LIN {X 177.96, Y 27.59, Z 0.00, A 0, B 0, C 0} C_DIS
LIN {X 177.78, Y 27.40, Z 0.00, A 0, B 0, C 0} C_DIS
LIN {X 177.60, Y 27.22, Z 0.00, A 0, B 0, C 0} C_DIS
LIN {X 177.41, Y 27.05, Z 0.00, A 0, B 0, C 0} C_DIS
LIN {X 177.23, Y 26.88, Z 0.00, A 0, B 0, C 0} C_DIS
LIN {X 177.05, Y 26.69, Z 0.00, A 0, B 0, C 0} C_DIS
LIN {X 176.88, Y 26.50, Z 0.00, A 0, B 0, C 0} C_DIS
LIN {X 176.71, Y 26.29, Z 0.00, A 0, B 0, C 0} C_DIS
LIN {X 176.55, Y 26.07, Z 0.00, A 0, B 0, C 0} C_DIS
LIN {X 176.39, Y 25.84, Z 0.00, A 0, B 0, C 0} C_DIS
LIN {X 176.24, Y 25.61, Z 0.00, A 0, B 0, C 0} C_DIS
LIN {X 176.09, Y 25.38, Z 0.00, A 0, B 0, C 0} C_DIS
LIN {X 175.93, Y 25.14, Z 0.00, A 0, B 0, C 0} C_DIS
LIN {X 175.78, Y 24.91, Z 0.00, A 0, B 0, C 0} C_DIS
LIN {X 175.63, Y 24.68, Z 0.00, A 0, B 0, C 0} C_DIS
LIN {X 175.47, Y 24.45, Z 0.00, A 0, B 0, C 0} C_DIS
LIN {X 175.32, Y 24.21, Z 0.00, A 0, B 0, C 0} C_DIS
LIN {X 175.17, Y 23.98, Z 0.00, A 0, B 0, C 0} C_DIS
LIN {X 175.01, Y 23.75, Z 0.00, A 0, B 0, C 0} C_DIS
LIN {X 174.86, Y 23.52, Z 0.00, A 0, B 0, C 0} C_DIS
LIN {X 174.71, Y 23.29, Z 0.00, A 0, B 0, C 0} C_DIS
LIN {X 174.55, Y 23.05, Z 0.00, A 0, B 0, C 0} C_DIS
LIN {X 174.40, Y 22.82, Z 0.00, A 0, B 0, C 0} C_DIS
LIN {X 174.24, Y 22.59, Z 0.00, A 0, B 0, C 0} C_DIS
LIN {X 174.09, Y 22.36, Z 0.00, A 0, B 0, C 0} C_DIS
LIN {X 173.94, Y 22.13, Z 0.00, A 0, B 0, C 0} C_DIS
LIN {X 173.78, Y 21.90, Z 0.00, A 0, B 0, C 0} C_DIS
LIN {X 173.63, Y 21.66, Z 0.00, A 0, B 0, C 0} C_DIS
LIN {X 173.48, Y 21.43, Z 0.00, A 0, B 0, C 0} C_DIS
LIN {X 173.32, Y 21.20, Z 0.00, A 0, B 0, C 0} C_DIS
LIN {X 173.17, Y 20.97, Z 0.00, A 0, B 0, C 0} C_DIS
LIN {X 173.01, Y 20.74, Z 0.00, A 0, B 0, C 0} C_DIS
LIN {X 172.86, Y 20.51, Z 0.00, A 0, B 0, C 0} C_DIS
LIN {X 172.71, Y 20.28, Z 0.00, A 0, B 0, C 0} C_DIS
LIN {X 172.55, Y 20.04, Z 0.00, A 0, B 0, C 0} C_DIS
LIN {X 172.40, Y 19.81, Z 0.00, A 0, B 0, C 0} C_DIS
LIN {X 172.24, Y 19.58, Z 0.00, A 0, B 0, C 0} C_DIS
LIN {X 172.09, Y 19.35, Z 0.00, A 0, B 0, C 0} C_DIS
LIN {X 171.94, Y 19.12, Z 0.00, A 0, B 0, C 0} C_DIS
LIN {X 171.78, Y 18.89, Z 0.00, A 0, B 0, C 0} C_DIS
LIN {X 171.63, Y 18.65, Z 0.00, A 0, B 0, C 0} C_DIS
LIN {X 171.48, Y 18.42, Z 0.00, A 0, B 0, C 0} C_DIS
LIN {X 171.32, Y 18.19, Z 0.00, A 0, B 0, C 0} C_DIS
LIN {X 171.17, Y 17.96, Z 0.00, A 0, B 0, C 0} C_DIS
LIN {X 171.01, Y 17.73, Z 0.00, A 0, B 0, C 0} C_DIS
LIN {X 170.86, Y 17.49, Z 0.00, A 0, B 0, C 0} C_DIS
LIN {X 170.71, Y 17.26, Z 0.00, A 0, B 0, C 0} C_DIS
LIN {X 170.55, Y 17.03, Z 0.00, A 0, B 0, C 0} C_DIS
LIN {X 170.40, Y 16.80, Z 0.00, A 0, B 0, C 0} C_DIS
LIN {X 170.25, Y 16.57, Z 0.00, A 0, B 0, C 0} C_DIS
LIN {X 170.09, Y 16.33, Z 0.00, A 0, B 0, C 0} C_DIS
LIN {X 169.94, Y 16.10, Z 0.00, A 0, B 0, C 0} C_DIS
LIN {X 169.78, Y 15.87, Z 0.00, A 0, B 0, C 0} C_DIS
LIN {X 169.63, Y 15.64, Z 0.00, A 0, B 0, C 0} C_DIS
LIN {X 169.48, Y 15.41, Z 0.00, A 0, B 0, C 0} C_DIS
LIN {X 169.32, Y 15.18, Z 0.00, A 0, B 0, C 0} C_DIS
LIN {X 169.17, Y 14.94, Z 0.00, A 0, B 0, C 0} C_DIS
LIN {X 169.02, Y 14.71, Z 0.00, A 0, B 0, C 0} C_DIS
LIN {X 168.86, Y 14.48, Z 0.00, A 0, B 0, C 0} C_DIS
LIN {X 168.71, Y 14.25, Z 0.00, A 0, B 0, C 0} C_DIS
LIN {X 168.55, Y 14.02, Z 0.00, A 0, B 0, C 0} C_DIS
LIN {X 168.40, Y 13.79, Z 0.00, A 0, B 0, C 0} C_DIS
LIN {X 168.25, Y 13.55, Z 0.00, A 0, B 0, C 0} C_DIS
LIN {X 168.09, Y 13.32, Z 0.00, A 0, B 0, C 0} C_DIS
LIN {X 167.94, Y 13.09, Z 0.00, A 0, B 0, C 0} C_DIS
LIN {X 167.79, Y 12.86, Z 0.00, A 0, B 0, C 0} C_DIS
LIN {X 167.63, Y 12.63, Z 0.00, A 0, B 0, C 0} C_DIS
LIN {X 167.48, Y 12.40, Z 0.00, A 0, B 0, C 0} C_DIS
LIN {X 167.32, Y 12.17, Z 0.00, A 0, B 0, C 0} C_DIS
LIN {X 167.17, Y 11.93, Z 0.00, A 0, B 0, C 0} C_DIS
LIN {X 167.02, Y 11.70, Z 0.00, A 0, B 0, C 0} C_DIS
LIN {X 166.86, Y 11.47, Z 0.00, A 0, B 0, C 0} C_DIS
LIN {X 166.71, Y 11.24, Z 0.00, A 0, B 0, C 0} C_DIS
LIN {X 166.55, Y 11.01, Z 0.00, A 0, B 0, C 0} C_DIS
LIN {X 166.40, Y 10.78, Z 0.00, A 0, B 0, C 0} C_DIS
LIN {X 166.25, Y 10.54, Z 0.00, A 0, B 0, C 0} C_DIS
LIN {X 166.09, Y 10.31, Z 0.00, A 0, B 0, C 0} C_DIS
LIN {X 165.94, Y 10.08, Z 0.00, A 0, B 0, C 0} C_DIS
LIN {X 165.79, Y 9.85, Z 0.00, A 0, B 0, C 0} C_DIS
LIN {X 165.63, Y 9.62, Z 0.00, A 0, B 0, C 0} C_DIS
LIN {X 165.48, Y 9.38, Z 0.00, A 0, B 0, C 0} C_DIS
LIN {X 165.33, Y 9.15, Z 0.00, A 0, B 0, C 0} C_DIS
LIN {X 165.17, Y 8.92, Z 0.00, A 0, B 0, C 0} C_DIS
LIN {X 165.02, Y 8.68, Z 0.00, A 0, B 0, C 0} C_DIS
LIN {X 164.87, Y 8.45, Z 0.00, A 0, B 0, C 0} C_DIS
LIN {X 164.71, Y 8.22, Z 0.00, A 0, B 0, C 0} C_DIS
LIN {X 164.56, Y 7.99, Z 0.00, A 0, B 0, C 0} C_DIS
LIN {X 164.40, Y 7.76, Z 0.00, A 0, B 0, C 0} C_DIS
LIN {X 164.24, Y 7.54, Z 0.00, A 0, B 0, C 0} C_DIS
LIN {X 164.08, Y 7.33, Z 0.00, A 0, B 0, C 0} C_DIS
LIN {X 163.91, Y 7.13, Z 0.00, A 0, B 0, C 0} C_DIS
LIN {X 163.73, Y 6.94, Z 0.00, A 0, B 0, C 0} C_DIS
LIN {X 163.54, Y 6.77, Z 0.00, A 0, B 0, C 0} C_DIS
LIN {X 163.36, Y 6.60, Z 0.00, A 0, B 0, C 0} C_DIS
LIN {X 163.17, Y 6.42, Z 0.00, A 0, B 0, C 0} C_DIS
LIN {X 163.00, Y 6.23, Z 0.00, A 0, B 0, C 0} C_DIS
LIN {X 162.83, Y 6.02, Z 0.00, A 0, B 0, C 0} C_DIS
LIN {X 162.67, Y 5.80, Z 0.00, A 0, B 0, C 0} C_DIS
LIN {X 162.51, Y 5.58, Z 0.00, A 0, B 0, C 0} C_DIS
LIN {X 162.34, Y 5.37, Z 0.00, A 0, B 0, C 0} C_DIS
LIN {X 162.17, Y 5.17, Z 0.00, A 0, B 0, C 0} C_DIS
LIN {X 162.00, Y 4.98, Z 0.00, A 0, B 0, C 0} C_DIS
LIN {X 161.81, Y 4.80, Z 0.00, A 0, B 0, C 0} C_DIS
LIN {X 161.62, Y 4.64, Z 0.00, A 0, B 0, C 0} C_DIS
LIN {X 161.43, Y 4.51, Z 0.00, A 0, B 0, C 0} C_DIS
LIN {X 161.23, Y 4.38, Z 0.00, A 0, B 0, C 0} C_DIS
LIN {X 161.03, Y 4.23, Z 0.00, A 0, B 0, C 0} C_DIS
LIN {X 160.84, Y 4.07, Z 0.00, A 0, B 0, C 0} C_DIS
LIN {X 160.66, Y 3.89, Z 0.00, A 0, B 0, C 0} C_DIS
LIN {X 160.48, Y 3.70, Z 0.00, A 0, B 0, C 0} C_DIS
LIN {X 160.30, Y 3.52, Z 0.00, A 0, B 0, C 0} C_DIS
LIN {X 160.12, Y 3.33, Z 0.00, A 0, B 0, C 0} C_DIS
LIN {X 159.94, Y 3.15, Z 0.00, A 0, B 0, C 0} C_DIS
LIN {X 159.76, Y 2.97, Z 0.00, A 0, B 0, C 0} C_DIS
LIN {X 159.58, Y 2.79, Z 0.00, A 0, B 0, C 0} C_DIS
LIN {X 159.39, Y 2.63, Z 0.00, A 0, B 0, C 0} C_DIS
LIN {X 159.20, Y 2.49, Z 0.00, A 0, B 0, C 0} C_DIS
LIN {X 158.99, Y 2.39, Z 0.00, A 0, B 0, C 0} C_DIS
LIN {X 158.78, Y 2.31, Z 0.00, A 0, B 0, C 0} C_DIS
LIN {X 158.56, Y 2.25, Z 0.00, A 0, B 0, C 0} C_DIS
LIN {X 158.35, Y 2.17, Z 0.00, A 0, B 0, C 0} C_DIS
LIN {X 158.14, Y 2.09, Z 0.00, A 0, B 0, C 0} C_DIS
LIN {X 157.93, Y 2.00, Z 0.00, A 0, B 0, C 0} C_DIS
LIN {X 157.72, Y 1.92, Z 0.00, A 0, B 0, C 0} C_DIS
LIN {X 157.51, Y 1.85, Z 0.00, A 0, B 0, C 0} C_DIS
LIN {X 157.30, Y 1.78, Z 0.00, A 0, B 0, C 0} C_DIS
LIN {X 157.09, Y 1.69, Z 0.00, A 0, B 0, C 0} C_DIS
LIN {X 156.88, Y 1.57, Z 0.00, A 0, B 0, C 0} C_DIS
LIN {X 156.69, Y 1.44, Z 0.00, A 0, B 0, C 0} C_DIS
LIN {X 156.49, Y 1.31, Z 0.00, A 0, B 0, C 0} C_DIS
LIN {X 156.28, Y 1.21, Z 0.00, A 0, B 0, C 0} C_DIS
LIN {X 156.07, Y 1.14, Z 0.00, A 0, B 0, C 0} C_DIS
LIN {X 155.85, Y 1.06, Z 0.00, A 0, B 0, C 0} C_DIS
LIN {X 155.64, Y 0.98, Z 0.00, A 0, B 0, C 0} C_DIS
LIN {X 155.43, Y 0.89, Z 0.00, A 0, B 0, C 0} C_DIS
LIN {X 155.22, Y 0.84, Z 0.00, A 0, B 0, C 0} C_DIS
LIN {X 155.00, Y 0.82, Z 0.00, A 0, B 0, C 0} C_DIS
LIN {X 154.79, Y 0.81, Z 0.00, A 0, B 0, C 0} C_DIS
LIN {X 154.57, Y 0.81, Z 0.00, A 0, B 0, C 0} C_DIS
LIN {X 154.35, Y 0.81, Z 0.00, A 0, B 0, C 0} C_DIS
LIN {X 154.13, Y 0.81, Z 0.00, A 0, B 0, C 0} C_DIS
LIN {X 153.92, Y 0.81, Z 0.00, A 0, B 0, C 0} C_DIS
LIN {X 153.70, Y 0.82, Z 0.00, A 0, B 0, C 0} C_DIS
LIN {X 153.48, Y 0.82, Z 0.00, A 0, B 0, C 0} C_DIS
LIN {X 153.26, Y 0.82, Z 0.00, A 0, B 0, C 0} C_DIS
LIN {X 153.05, Y 0.81, Z 0.00, A 0, B 0, C 0} C_DIS
LIN {X 152.83, Y 0.81, Z 0.00, A 0, B 0, C 0} C_DIS
LIN {X 152.61, Y 0.81, Z 0.00, A 0, B 0, C 0} C_DIS
LIN {X 152.39, Y 0.81, Z 0.00, A 0, B 0, C 0} C_DIS
LIN {X 152.18, Y 0.81, Z 0.00, A 0, B 0, C 0} C_DIS
LIN {X 151.96, Y 0.81, Z 0.00, A 0, B 0, C 0} C_DIS
LIN {X 151.74, Y 0.81, Z 0.00, A 0, B 0, C 0} C_DIS
LIN {X 151.52, Y 0.81, Z 0.00, A 0, B 0, C 0} C_DIS
LIN {X 151.31, Y 0.81, Z 0.00, A 0, B 0, C 0} C_DIS
LIN {X 151.09, Y 0.81, Z 0.00, A 0, B 0, C 0} C_DIS
LIN {X 150.87, Y 0.81, Z 0.00, A 0, B 0, C 0} C_DIS
LIN {X 150.65, Y 0.81, Z 0.00, A 0, B 0, C 0} C_DIS
LIN {X 150.44, Y 0.81, Z 0.00, A 0, B 0, C 0} C_DIS
LIN {X 150.22, Y 0.81, Z 0.00, A 0, B 0, C 0} C_DIS
LIN {X 150.00, Y 0.81, Z 0.00, A 0, B 0, C 0} C_DIS
LIN {X 149.78, Y 0.81, Z 0.00, A 0, B 0, C 0} C_DIS
LIN {X 149.57, Y 0.81, Z 0.00, A 0, B 0, C 0} C_DIS
LIN {X 149.35, Y 0.81, Z 0.00, A 0, B 0, C 0} C_DIS
LIN {X 149.13, Y 0.81, Z 0.00, A 0, B 0, C 0} C_DIS
LIN {X 148.91, Y 0.81, Z 0.00, A 0, B 0, C 0} C_DIS
LIN {X 148.70, Y 0.81, Z 0.00, A 0, B 0, C 0} C_DIS
LIN {X 148.48, Y 0.81, Z 0.00, A 0, B 0, C 0} C_DIS
LIN {X 148.26, Y 0.81, Z 0.00, A 0, B 0, C 0} C_DIS
LIN {X 148.04, Y 0.81, Z 0.00, A 0, B 0, C 0} C_DIS
LIN {X 147.83, Y 0.81, Z 0.00, A 0, B 0, C 0} C_DIS
LIN {X 147.61, Y 0.81, Z 0.00, A 0, B 0, C 0} C_DIS
LIN {X 147.39, Y 0.81, Z 0.00, A 0, B 0, C 0} C_DIS
LIN {X 147.17, Y 0.81, Z 0.00, A 0, B 0, C 0} C_DIS
LIN {X 146.96, Y 0.81, Z 0.00, A 0, B 0, C 0} C_DIS
LIN {X 146.74, Y 0.81, Z 0.00, A 0, B 0, C 0} C_DIS
LIN {X 146.52, Y 0.81, Z 0.00, A 0, B 0, C 0} C_DIS
LIN {X 146.30, Y 0.81, Z 0.00, A 0, B 0, C 0} C_DIS
LIN {X 146.09, Y 0.81, Z 0.00, A 0, B 0, C 0} C_DIS
LIN {X 145.87, Y 0.81, Z 0.00, A 0, B 0, C 0} C_DIS
LIN {X 145.65, Y 0.81, Z 0.00, A 0, B 0, C 0} C_DIS
LIN {X 145.43, Y 0.81, Z 0.00, A 0, B 0, C 0} C_DIS
LIN {X 145.22, Y 0.81, Z 0.00, A 0, B 0, C 0} C_DIS
LIN {X 145.00, Y 0.81, Z 0.00, A 0, B 0, C 0} C_DIS
LIN {X 144.78, Y 0.81, Z 0.00, A 0, B 0, C 0} C_DIS
LIN {X 144.56, Y 0.81, Z 0.00, A 0, B 0, C 0} C_DIS
LIN {X 144.35, Y 0.81, Z 0.00, A 0, B 0, C 0} C_DIS
LIN {X 144.13, Y 0.81, Z 0.00, A 0, B 0, C 0} C_DIS
LIN {X 143.91, Y 0.81, Z 0.00, A 0, B 0, C 0} C_DIS
LIN {X 143.69, Y 0.81, Z 0.00, A 0, B 0, C 0} C_DIS
LIN {X 143.48, Y 0.81, Z 0.00, A 0, B 0, C 0} C_DIS
LIN {X 143.26, Y 0.81, Z 0.00, A 0, B 0, C 0} C_DIS
LIN {X 143.04, Y 0.81, Z 0.00, A 0, B 0, C 0} C_DIS
LIN {X 142.83, Y 0.81, Z 0.00, A 0, B 0, C 0} C_DIS
LIN {X 142.61, Y 0.81, Z 0.00, A 0, B 0, C 0} C_DIS
LIN {X 142.39, Y 0.81, Z 0.00, A 0, B 0, C 0} C_DIS
LIN {X 142.17, Y 0.81, Z 0.00, A 0, B 0, C 0} C_DIS
LIN {X 141.96, Y 0.81, Z 0.00, A 0, B 0, C 0} C_DIS
LIN {X 141.74, Y 0.81, Z 0.00, A 0, B 0, C 0} C_DIS
LIN {X 141.52, Y 0.81, Z 0.00, A 0, B 0, C 0} C_DIS
LIN {X 141.30, Y 0.81, Z 0.00, A 0, B 0, C 0} C_DIS
LIN {X 141.09, Y 0.81, Z 0.00, A 0, B 0, C 0} C_DIS
LIN {X 140.87, Y 0.81, Z 0.00, A 0, B 0, C 0} C_DIS
LIN {X 140.65, Y 0.81, Z 0.00, A 0, B 0, C 0} C_DIS
LIN {X 140.43, Y 0.81, Z 0.00, A 0, B 0, C 0} C_DIS
LIN {X 140.22, Y 0.81, Z 0.00, A 0, B 0, C 0} C_DIS
LIN {X 140.00, Y 0.81, Z 0.00, A 0, B 0, C 0} C_DIS
LIN {X 139.78, Y 0.81, Z 0.00, A 0, B 0, C 0} C_DIS
LIN {X 139.56, Y 0.81, Z 0.00, A 0, B 0, C 0} C_DIS
LIN {X 139.35, Y 0.81, Z 0.00, A 0, B 0, C 0} C_DIS
LIN {X 139.13, Y 0.81, Z 0.00, A 0, B 0, C 0} C_DIS
LIN {X 138.91, Y 0.81, Z 0.00, A 0, B 0, C 0} C_DIS
LIN {X 138.69, Y 0.81, Z 0.00, A 0, B 0, C 0} C_DIS
LIN {X 138.48, Y 0.81, Z 0.00, A 0, B 0, C 0} C_DIS
LIN {X 138.26, Y 0.81, Z 0.00, A 0, B 0, C 0} C_DIS
LIN {X 138.04, Y 0.81, Z 0.00, A 0, B 0, C 0} C_DIS
LIN {X 137.82, Y 0.81, Z 0.00, A 0, B 0, C 0} C_DIS
LIN {X 137.61, Y 0.81, Z 0.00, A 0, B 0, C 0} C_DIS
LIN {X 137.39, Y 0.81, Z 0.00, A 0, B 0, C 0} C_DIS
LIN {X 137.17, Y 0.81, Z 0.00, A 0, B 0, C 0} C_DIS
LIN {X 136.95, Y 0.81, Z 0.00, A 0, B 0, C 0} C_DIS
LIN {X 136.74, Y 0.81, Z 0.00, A 0, B 0, C 0} C_DIS
LIN {X 136.52, Y 0.81, Z 0.00, A 0, B 0, C 0} C_DIS
LIN {X 136.30, Y 0.81, Z 0.00, A 0, B 0, C 0} C_DIS
LIN {X 136.08, Y 0.81, Z 0.00, A 0, B 0, C 0} C_DIS
LIN {X 135.87, Y 0.81, Z 0.00, A 0, B 0, C 0} C_DIS
LIN {X 135.65, Y 0.81, Z 0.00, A 0, B 0, C 0} C_DIS
LIN {X 135.43, Y 0.82, Z 0.00, A 0, B 0, C 0} C_DIS
LIN {X 135.21, Y 0.82, Z 0.00, A 0, B 0, C 0} C_DIS
LIN {X 135.00, Y 0.81, Z 0.00, A 0, B 0, C 0} C_DIS
LIN {X 134.78, Y 0.81, Z 0.00, A 0, B 0, C 0} C_DIS
LIN {X 134.56, Y 0.81, Z 0.00, A 0, B 0, C 0} C_DIS
LIN {X 134.34, Y 0.81, Z 0.00, A 0, B 0, C 0} C_DIS
LIN {X 134.13, Y 0.80, Z 0.00, A 0, B 0, C 0} C_DIS
LIN {X 133.91, Y 0.81, Z 0.00, A 0, B 0, C 0} C_DIS
LIN {X 133.69, Y 0.82, Z 0.00, A 0, B 0, C 0} C_DIS
LIN {X 133.48, Y 0.85, Z 0.00, A 0, B 0, C 0} C_DIS
LIN {X 133.26, Y 0.90, Z 0.00, A 0, B 0, C 0} C_DIS
LIN {X 133.05, Y 0.98, Z 0.00, A 0, B 0, C 0} C_DIS
LIN {X 132.84, Y 1.06, Z 0.00, A 0, B 0, C 0} C_DIS
LIN {X 132.63, Y 1.14, Z 0.00, A 0, B 0, C 0} C_DIS
LIN {X 132.42, Y 1.26, Z 0.00, A 0, B 0, C 0} C_DIS
LIN {X 132.24, Y 1.42, Z 0.00, A 0, B 0, C 0} C_DIS
LIN {X 132.08, Y 1.65, Z 0.00, A 0, B 0, C 0} C_DIS
LIN {X 131.93, Y 1.89, Z 0.00, A 0, B 0, C 0} C_DIS
LIN {X 131.78, Y 2.13, Z 0.00, A 0, B 0, C 0} C_DIS
LIN {X 131.64, Y 2.37, Z 0.00, A 0, B 0, C 0} C_DIS
LIN {X 131.53, Y 2.64, Z 0.00, A 0, B 0, C 0} C_DIS
LIN {X 131.45, Y 2.95, Z 0.00, A 0, B 0, C 0} C_DIS
LIN {X 131.40, Y 3.28, Z 0.00, A 0, B 0, C 0} C_DIS
LIN {X 131.36, Y 3.60, Z 0.00, A 0, B 0, C 0} C_DIS
LIN {X 131.32, Y 3.93, Z 0.00, A 0, B 0, C 0} C_DIS
LIN {X 131.29, Y 4.25, Z 0.00, A 0, B 0, C 0} C_DIS
LIN {X 131.27, Y 4.57, Z 0.00, A 0, B 0, C 0} C_DIS
LIN {X 131.26, Y 4.89, Z 0.00, A 0, B 0, C 0} C_DIS
LIN {X 131.25, Y 5.22, Z 0.00, A 0, B 0, C 0} C_DIS
LIN {X 131.25, Y 5.55, Z 0.00, A 0, B 0, C 0} C_DIS
LIN {X 131.25, Y 5.88, Z 0.00, A 0, B 0, C 0} C_DIS
LIN {X 131.26, Y 6.21, Z 0.00, A 0, B 0, C 0} C_DIS
LIN {X 131.26, Y 6.53, Z 0.00, A 0, B 0, C 0} C_DIS
LIN {X 131.26, Y 6.86, Z 0.00, A 0, B 0, C 0} C_DIS
LIN {X 131.26, Y 7.19, Z 0.00, A 0, B 0, C 0} C_DIS
LIN {X 131.26, Y 7.52, Z 0.00, A 0, B 0, C 0} C_DIS
LIN {X 131.26, Y 7.85, Z 0.00, A 0, B 0, C 0} C_DIS
LIN {X 131.26, Y 8.17, Z 0.00, A 0, B 0, C 0} C_DIS
LIN {X 131.26, Y 8.50, Z 0.00, A 0, B 0, C 0} C_DIS
LIN {X 131.26, Y 8.83, Z 0.00, A 0, B 0, C 0} C_DIS
LIN {X 131.26, Y 9.16, Z 0.00, A 0, B 0, C 0} C_DIS
LIN {X 131.26, Y 9.49, Z 0.00, A 0, B 0, C 0} C_DIS
LIN {X 131.26, Y 9.81, Z 0.00, A 0, B 0, C 0} C_DIS
LIN {X 131.26, Y 10.14, Z 0.00, A 0, B 0, C 0} C_DIS
LIN {X 131.26, Y 10.47, Z 0.00, A 0, B 0, C 0} C_DIS
LIN {X 131.26, Y 10.80, Z 0.00, A 0, B 0, C 0} C_DIS
LIN {X 131.26, Y 11.12, Z 0.00, A 0, B 0, C 0} C_DIS
LIN {X 131.26, Y 11.45, Z 0.00, A 0, B 0, C 0} C_DIS
LIN {X 131.26, Y 11.78, Z 0.00, A 0, B 0, C 0} C_DIS
LIN {X 131.26, Y 12.11, Z 0.00, A 0, B 0, C 0} C_DIS
LIN {X 131.26, Y 12.43, Z 0.00, A 0, B 0, C 0} C_DIS
LIN {X 131.26, Y 12.76, Z 0.00, A 0, B 0, C 0} C_DIS
LIN {X 131.26, Y 13.09, Z 0.00, A 0, B 0, C 0} C_DIS
LIN {X 131.26, Y 13.42, Z 0.00, A 0, B 0, C 0} C_DIS
LIN {X 131.26, Y 13.75, Z 0.00, A 0, B 0, C 0} C_DIS
LIN {X 131.26, Y 14.07, Z 0.00, A 0, B 0, C 0} C_DIS
LIN {X 131.26, Y 14.40, Z 0.00, A 0, B 0, C 0} C_DIS
LIN {X 131.26, Y 14.73, Z 0.00, A 0, B 0, C 0} C_DIS
LIN {X 131.26, Y 15.06, Z 0.00, A 0, B 0, C 0} C_DIS
LIN {X 131.26, Y 15.38, Z 0.00, A 0, B 0, C 0} C_DIS
LIN {X 131.26, Y 15.71, Z 0.00, A 0, B 0, C 0} C_DIS
LIN {X 131.26, Y 16.04, Z 0.00, A 0, B 0, C 0} C_DIS
LIN {X 131.26, Y 16.37, Z 0.00, A 0, B 0, C 0} C_DIS
LIN {X 131.26, Y 16.69, Z 0.00, A 0, B 0, C 0} C_DIS
LIN {X 131.26, Y 17.02, Z 0.00, A 0, B 0, C 0} C_DIS
LIN {X 131.26, Y 17.35, Z 0.00, A 0, B 0, C 0} C_DIS
LIN {X 131.26, Y 17.68, Z 0.00, A 0, B 0, C 0} C_DIS
LIN {X 131.26, Y 18.01, Z 0.00, A 0, B 0, C 0} C_DIS
LIN {X 131.26, Y 18.33, Z 0.00, A 0, B 0, C 0} C_DIS
LIN {X 131.26, Y 18.66, Z 0.00, A 0, B 0, C 0} C_DIS
LIN {X 131.26, Y 18.99, Z 0.00, A 0, B 0, C 0} C_DIS
LIN {X 131.26, Y 19.32, Z 0.00, A 0, B 0, C 0} C_DIS
LIN {X 131.26, Y 19.64, Z 0.00, A 0, B 0, C 0} C_DIS
LIN {X 131.26, Y 19.97, Z 0.00, A 0, B 0, C 0} C_DIS
LIN {X 131.26, Y 20.30, Z 0.00, A 0, B 0, C 0} C_DIS
LIN {X 131.26, Y 20.63, Z 0.00, A 0, B 0, C 0} C_DIS
LIN {X 131.26, Y 20.95, Z 0.00, A 0, B 0, C 0} C_DIS
LIN {X 131.26, Y 21.28, Z 0.00, A 0, B 0, C 0} C_DIS
LIN {X 131.26, Y 21.61, Z 0.00, A 0, B 0, C 0} C_DIS
LIN {X 131.26, Y 21.94, Z 0.00, A 0, B 0, C 0} C_DIS
LIN {X 131.26, Y 22.27, Z 0.00, A 0, B 0, C 0} C_DIS
LIN {X 131.26, Y 22.59, Z 0.00, A 0, B 0, C 0} C_DIS
LIN {X 131.26, Y 22.92, Z 0.00, A 0, B 0, C 0} C_DIS
LIN {X 131.26, Y 23.25, Z 0.00, A 0, B 0, C 0} C_DIS
LIN {X 131.26, Y 23.58, Z 0.00, A 0, B 0, C 0} C_DIS
LIN {X 131.26, Y 23.90, Z 0.00, A 0, B 0, C 0} C_DIS
LIN {X 131.26, Y 24.23, Z 0.00, A 0, B 0, C 0} C_DIS
LIN {X 131.26, Y 24.56, Z 0.00, A 0, B 0, C 0} C_DIS
LIN {X 131.26, Y 24.89, Z 0.00, A 0, B 0, C 0} C_DIS
LIN {X 131.26, Y 25.21, Z 0.00, A 0, B 0, C 0} C_DIS
LIN {X 131.26, Y 25.54, Z 0.00, A 0, B 0, C 0} C_DIS
LIN {X 131.26, Y 25.87, Z 0.00, A 0, B 0, C 0} C_DIS
LIN {X 131.26, Y 26.20, Z 0.00, A 0, B 0, C 0} C_DIS
LIN {X 131.26, Y 26.53, Z 0.00, A 0, B 0, C 0} C_DIS
LIN {X 131.26, Y 26.85, Z 0.00, A 0, B 0, C 0} C_DIS
LIN {X 131.26, Y 27.18, Z 0.00, A 0, B 0, C 0} C_DIS
LIN {X 131.26, Y 27.51, Z 0.00, A 0, B 0, C 0} C_DIS
LIN {X 131.26, Y 27.84, Z 0.00, A 0, B 0, C 0} C_DIS
LIN {X 131.26, Y 28.16, Z 0.00, A 0, B 0, C 0} C_DIS
LIN {X 131.26, Y 28.49, Z 0.00, A 0, B 0, C 0} C_DIS
LIN {X 131.26, Y 28.82, Z 0.00, A 0, B 0, C 0} C_DIS
LIN {X 131.26, Y 29.15, Z 0.00, A 0, B 0, C 0} C_DIS
LIN {X 131.26, Y 29.48, Z 0.00, A 0, B 0, C 0} C_DIS
LIN {X 131.26, Y 29.80, Z 0.00, A 0, B 0, C 0} C_DIS
LIN {X 131.26, Y 30.13, Z 0.00, A 0, B 0, C 0} C_DIS
LIN {X 131.26, Y 30.46, Z 0.00, A 0, B 0, C 0} C_DIS
LIN {X 131.26, Y 30.79, Z 0.00, A 0, B 0, C 0} C_DIS
LIN {X 131.26, Y 31.11, Z 0.00, A 0, B 0, C 0} C_DIS
LIN {X 131.26, Y 31.44, Z 0.00, A 0, B 0, C 0} C_DIS
LIN {X 131.26, Y 31.77, Z 0.00, A 0, B 0, C 0} C_DIS
LIN {X 131.26, Y 32.10, Z 0.00, A 0, B 0, C 0} C_DIS
LIN {X 131.26, Y 32.42, Z 0.00, A 0, B 0, C 0} C_DIS
LIN {X 131.26, Y 32.75, Z 0.00, A 0, B 0, C 0} C_DIS
LIN {X 131.26, Y 33.08, Z 0.00, A 0, B 0, C 0} C_DIS
LIN {X 131.26, Y 33.41, Z 0.00, A 0, B 0, C 0} C_DIS
LIN {X 131.26, Y 33.74, Z 0.00, A 0, B 0, C 0} C_DIS
LIN {X 131.26, Y 34.06, Z 0.00, A 0, B 0, C 0} C_DIS
LIN {X 131.26, Y 34.39, Z 0.00, A 0, B 0, C 0} C_DIS
LIN {X 131.26, Y 34.72, Z 0.00, A 0, B 0, C 0} C_DIS
LIN {X 131.26, Y 35.05, Z 0.00, A 0, B 0, C 0} C_DIS
LIN {X 131.26, Y 35.37, Z 0.00, A 0, B 0, C 0} C_DIS
LIN {X 131.26, Y 35.70, Z 0.00, A 0, B 0, C 0} C_DIS
LIN {X 131.26, Y 36.03, Z 0.00, A 0, B 0, C 0} C_DIS
LIN {X 131.26, Y 36.36, Z 0.00, A 0, B 0, C 0} C_DIS
LIN {X 131.26, Y 36.69, Z 0.00, A 0, B 0, C 0} C_DIS
LIN {X 131.26, Y 37.01, Z 0.00, A 0, B 0, C 0} C_DIS
LIN {X 131.26, Y 37.34, Z 0.00, A 0, B 0, C 0} C_DIS
LIN {X 131.26, Y 37.67, Z 0.00, A 0, B 0, C 0} C_DIS
LIN {X 131.26, Y 38.00, Z 0.00, A 0, B 0, C 0} C_DIS
LIN {X 131.26, Y 38.32, Z 0.00, A 0, B 0, C 0} C_DIS
LIN {X 131.26, Y 38.65, Z 0.00, A 0, B 0, C 0} C_DIS
LIN {X 131.26, Y 38.98, Z 0.00, A 0, B 0, C 0} C_DIS
LIN {X 131.26, Y 39.31, Z 0.00, A 0, B 0, C 0} C_DIS
LIN {X 131.26, Y 39.63, Z 0.00, A 0, B 0, C 0} C_DIS
LIN {X 131.26, Y 39.96, Z 0.00, A 0, B 0, C 0} C_DIS
LIN {X 131.26, Y 40.29, Z 0.00, A 0, B 0, C 0} C_DIS
LIN {X 131.26, Y 40.62, Z 0.00, A 0, B 0, C 0} C_DIS
LIN {X 131.26, Y 40.95, Z 0.00, A 0, B 0, C 0} C_DIS
LIN {X 131.26, Y 41.27, Z 0.00, A 0, B 0, C 0} C_DIS
LIN {X 131.26, Y 41.60, Z 0.00, A 0, B 0, C 0} C_DIS
LIN {X 131.26, Y 41.93, Z 0.00, A 0, B 0, C 0} C_DIS
LIN {X 131.26, Y 42.26, Z 0.00, A 0, B 0, C 0} C_DIS
LIN {X 131.26, Y 42.58, Z 0.00, A 0, B 0, C 0} C_DIS
LIN {X 131.26, Y 42.91, Z 0.00, A 0, B 0, C 0} C_DIS
LIN {X 131.26, Y 43.24, Z 0.00, A 0, B 0, C 0} C_DIS
LIN {X 131.26, Y 43.57, Z 0.00, A 0, B 0, C 0} C_DIS
LIN {X 131.26, Y 43.89, Z 0.00, A 0, B 0, C 0} C_DIS
LIN {X 131.26, Y 44.22, Z 0.00, A 0, B 0, C 0} C_DIS
LIN {X 131.26, Y 44.55, Z 0.00, A 0, B 0, C 0} C_DIS
LIN {X 131.26, Y 44.88, Z 0.00, A 0, B 0, C 0} C_DIS
LIN {X 131.26, Y 45.21, Z 0.00, A 0, B 0, C 0} C_DIS
LIN {X 131.26, Y 45.53, Z 0.00, A 0, B 0, C 0} C_DIS
LIN {X 131.26, Y 45.86, Z 0.00, A 0, B 0, C 0} C_DIS
LIN {X 131.26, Y 46.19, Z 0.00, A 0, B 0, C 0} C_DIS
LIN {X 131.26, Y 46.52, Z 0.00, A 0, B 0, C 0} C_DIS
LIN {X 131.26, Y 46.84, Z 0.00, A 0, B 0, C 0} C_DIS
LIN {X 131.26, Y 47.17, Z 0.00, A 0, B 0, C 0} C_DIS
LIN {X 131.26, Y 47.50, Z 0.00, A 0, B 0, C 0} C_DIS
LIN {X 131.26, Y 47.83, Z 0.00, A 0, B 0, C 0} C_DIS
LIN {X 131.26, Y 48.16, Z 0.00, A 0, B 0, C 0} C_DIS
LIN {X 131.26, Y 48.48, Z 0.00, A 0, B 0, C 0} C_DIS
LIN {X 131.26, Y 48.81, Z 0.00, A 0, B 0, C 0} C_DIS
LIN {X 131.26, Y 49.14, Z 0.00, A 0, B 0, C 0} C_DIS
LIN {X 131.26, Y 49.47, Z 0.00, A 0, B 0, C 0} C_DIS
LIN {X 131.26, Y 49.79, Z 0.00, A 0, B 0, C 0} C_DIS
LIN {X 131.26, Y 50.12, Z 0.00, A 0, B 0, C 0} C_DIS
LIN {X 131.26, Y 50.45, Z 0.00, A 0, B 0, C 0} C_DIS
LIN {X 131.26, Y 50.78, Z 0.00, A 0, B 0, C 0} C_DIS
LIN {X 131.26, Y 51.10, Z 0.00, A 0, B 0, C 0} C_DIS
LIN {X 131.26, Y 51.43, Z 0.00, A 0, B 0, C 0} C_DIS
LIN {X 131.26, Y 51.76, Z 0.00, A 0, B 0, C 0} C_DIS
LIN {X 131.26, Y 52.09, Z 0.00, A 0, B 0, C 0} C_DIS
LIN {X 131.26, Y 52.42, Z 0.00, A 0, B 0, C 0} C_DIS
LIN {X 131.26, Y 52.74, Z 0.00, A 0, B 0, C 0} C_DIS
LIN {X 131.26, Y 53.07, Z 0.00, A 0, B 0, C 0} C_DIS
LIN {X 131.26, Y 53.40, Z 0.00, A 0, B 0, C 0} C_DIS
LIN {X 131.26, Y 53.73, Z 0.00, A 0, B 0, C 0} C_DIS
LIN {X 131.26, Y 54.05, Z 0.00, A 0, B 0, C 0} C_DIS
LIN {X 131.26, Y 54.38, Z 0.00, A 0, B 0, C 0} C_DIS
LIN {X 131.26, Y 54.71, Z 0.00, A 0, B 0, C 0} C_DIS
LIN {X 131.26, Y 55.04, Z 0.00, A 0, B 0, C 0} C_DIS
LIN {X 131.26, Y 55.36, Z 0.00, A 0, B 0, C 0} C_DIS
LIN {X 131.26, Y 55.69, Z 0.00, A 0, B 0, C 0} C_DIS
LIN {X 131.26, Y 56.02, Z 0.00, A 0, B 0, C 0} C_DIS
LIN {X 131.26, Y 56.35, Z 0.00, A 0, B 0, C 0} C_DIS
LIN {X 131.26, Y 56.68, Z 0.00, A 0, B 0, C 0} C_DIS
LIN {X 131.26, Y 57.00, Z 0.00, A 0, B 0, C 0} C_DIS
LIN {X 131.26, Y 57.33, Z 0.00, A 0, B 0, C 0} C_DIS
LIN {X 131.26, Y 57.66, Z 0.00, A 0, B 0, C 0} C_DIS
LIN {X 131.26, Y 57.99, Z 0.00, A 0, B 0, C 0} C_DIS
LIN {X 131.26, Y 58.31, Z 0.00, A 0, B 0, C 0} C_DIS
LIN {X 131.26, Y 58.64, Z 0.00, A 0, B 0, C 0} C_DIS
LIN {X 131.26, Y 58.97, Z 0.00, A 0, B 0, C 0} C_DIS
LIN {X 131.26, Y 59.30, Z 0.00, A 0, B 0, C 0} C_DIS
LIN {X 131.26, Y 59.63, Z 0.00, A 0, B 0, C 0} C_DIS
LIN {X 131.27, Y 59.95, Z 0.00, A 0, B 0, C 0} C_DIS
LIN {X 131.27, Y 60.28, Z 0.00, A 0, B 0, C 0} C_DIS
LIN {X 131.27, Y 60.61, Z 0.00, A 0, B 0, C 0} C_DIS
LIN {X 131.27, Y 60.94, Z 0.00, A 0, B 0, C 0} C_DIS
LIN {X 131.27, Y 61.26, Z 0.00, A 0, B 0, C 0} C_DIS
LIN {X 131.26, Y 61.59, Z 0.00, A 0, B 0, C 0} C_DIS
LIN {X 131.25, Y 61.92, Z 0.00, A 0, B 0, C 0} C_DIS
LIN {X 131.24, Y 62.25, Z 0.00, A 0, B 0, C 0} C_DIS
LIN {X 131.23, Y 62.57, Z 0.00, A 0, B 0, C 0} C_DIS
LIN {X 131.20, Y 62.90, Z 0.00, A 0, B 0, C 0} C_DIS
LIN {X 131.16, Y 63.22, Z 0.00, A 0, B 0, C 0} C_DIS
LIN {X 131.11, Y 63.53, Z 0.00, A 0, B 0, C 0} C_DIS
LIN {X 131.04, Y 63.85, Z 0.00, A 0, B 0, C 0} C_DIS
LIN {X 130.98, Y 64.17, Z 0.00, A 0, B 0, C 0} C_DIS
LIN {X 130.93, Y 64.48, Z 0.00, A 0, B 0, C 0} C_DIS
LIN {X 130.88, Y 64.80, Z 0.00, A 0, B 0, C 0} C_DIS
LIN {X 130.85, Y 65.13, Z 0.00, A 0, B 0, C 0} C_DIS
LIN {X 130.83, Y 65.45, Z 0.00, A 0, B 0, C 0} C_DIS
LIN {X 130.82, Y 65.78, Z 0.00, A 0, B 0, C 0} C_DIS
LIN {X 130.82, Y 66.11, Z 0.00, A 0, B 0, C 0} C_DIS
LIN {X 130.82, Y 66.43, Z 0.00, A 0, B 0, C 0} C_DIS
LIN {X 130.83, Y 66.76, Z 0.00, A 0, B 0, C 0} C_DIS
LIN {X 130.83, Y 67.09, Z 0.00, A 0, B 0, C 0} C_DIS
LIN {X 130.84, Y 67.42, Z 0.00, A 0, B 0, C 0} C_DIS
LIN {X 130.83, Y 67.75, Z 0.00, A 0, B 0, C 0} C_DIS
LIN {X 130.82, Y 68.07, Z 0.00, A 0, B 0, C 0} C_DIS
LIN {X 130.80, Y 68.40, Z 0.00, A 0, B 0, C 0} C_DIS
LIN {X 130.77, Y 68.72, Z 0.00, A 0, B 0, C 0} C_DIS
LIN {X 130.73, Y 69.04, Z 0.00, A 0, B 0, C 0} C_DIS
LIN {X 130.68, Y 69.36, Z 0.00, A 0, B 0, C 0} C_DIS
LIN {X 130.63, Y 69.68, Z 0.00, A 0, B 0, C 0} C_DIS
LIN {X 130.57, Y 70.00, Z 0.00, A 0, B 0, C 0} C_DIS
LIN {X 130.51, Y 70.31, Z 0.00, A 0, B 0, C 0} C_DIS
LIN {X 130.46, Y 70.63, Z 0.00, A 0, B 0, C 0} C_DIS
LIN {X 130.40, Y 70.95, Z 0.00, A 0, B 0, C 0} C_DIS
LIN {X 130.35, Y 71.27, Z 0.00, A 0, B 0, C 0} C_DIS
LIN {X 130.30, Y 71.59, Z 0.00, A 0, B 0, C 0} C_DIS
LIN {X 130.25, Y 71.90, Z 0.00, A 0, B 0, C 0} C_DIS
LIN {X 130.20, Y 72.22, Z 0.00, A 0, B 0, C 0} C_DIS
LIN {X 130.15, Y 72.54, Z 0.00, A 0, B 0, C 0} C_DIS
LIN {X 130.08, Y 72.85, Z 0.00, A 0, B 0, C 0} C_DIS
LIN {X 130.01, Y 73.16, Z 0.00, A 0, B 0, C 0} C_DIS
LIN {X 129.92, Y 73.46, Z 0.00, A 0, B 0, C 0} C_DIS
LIN {X 129.83, Y 73.76, Z 0.00, A 0, B 0, C 0} C_DIS
LIN {X 129.78, Y 74.08, Z 0.00, A 0, B 0, C 0} C_DIS
LIN {X 129.72, Y 74.39, Z 0.00, A 0, B 0, C 0} C_DIS
LIN {X 129.63, Y 74.69, Z 0.00, A 0, B 0, C 0} C_DIS
LIN {X 129.52, Y 74.97, Z 0.00, A 0, B 0, C 0} C_DIS
LIN {X 129.40, Y 75.25, Z 0.00, A 0, B 0, C 0} C_DIS
LIN {X 129.32, Y 75.55, Z 0.00, A 0, B 0, C 0} C_DIS
LIN {X 129.27, Y 75.87, Z 0.00, A 0, B 0, C 0} C_DIS
LIN {X 129.21, Y 76.19, Z 0.00, A 0, B 0, C 0} C_DIS
LIN {X 129.12, Y 76.49, Z 0.00, A 0, B 0, C 0} C_DIS
LIN {X 129.03, Y 76.78, Z 0.00, A 0, B 0, C 0} C_DIS
LIN {X 128.95, Y 77.09, Z 0.00, A 0, B 0, C 0} C_DIS
LIN {X 128.90, Y 77.41, Z 0.00, A 0, B 0, C 0} C_DIS
LIN {X 128.84, Y 77.72, Z 0.00, A 0, B 0, C 0} C_DIS
LIN {X 128.75, Y 78.02, Z 0.00, A 0, B 0, C 0} C_DIS
LIN {X 128.63, Y 78.29, Z 0.00, A 0, B 0, C 0} C_DIS
LIN {X 128.52, Y 78.58, Z 0.00, A 0, B 0, C 0} C_DIS
LIN {X 128.44, Y 78.88, Z 0.00, A 0, B 0, C 0} C_DIS
LIN {X 128.35, Y 79.18, Z 0.00, A 0, B 0, C 0} C_DIS
LIN {X 128.25, Y 79.47, Z 0.00, A 0, B 0, C 0} C_DIS
LIN {X 128.14, Y 79.75, Z 0.00, A 0, B 0, C 0} C_DIS
LIN {X 128.02, Y 80.02, Z 0.00, A 0, B 0, C 0} C_DIS
LIN {X 127.89, Y 80.29, Z 0.00, A 0, B 0, C 0} C_DIS
LIN {X 127.76, Y 80.56, Z 0.00, A 0, B 0, C 0} C_DIS
LIN {X 127.64, Y 80.83, Z 0.00, A 0, B 0, C 0} C_DIS
LIN {X 127.52, Y 81.10, Z 0.00, A 0, B 0, C 0} C_DIS
LIN {X 127.40, Y 81.38, Z 0.00, A 0, B 0, C 0} C_DIS
LIN {X 127.30, Y 81.66, Z 0.00, A 0, B 0, C 0} C_DIS
LIN {X 127.20, Y 81.95, Z 0.00, A 0, B 0, C 0} C_DIS
LIN {X 127.11, Y 82.25, Z 0.00, A 0, B 0, C 0} C_DIS
LIN {X 127.01, Y 82.54, Z 0.00, A 0, B 0, C 0} C_DIS
LIN {X 126.91, Y 82.83, Z 0.00, A 0, B 0, C 0} C_DIS
LIN {X 126.80, Y 83.11, Z 0.00, A 0, B 0, C 0} C_DIS
LIN {X 126.68, Y 83.38, Z 0.00, A 0, B 0, C 0} C_DIS
LIN {X 126.54, Y 83.64, Z 0.00, A 0, B 0, C 0} C_DIS
LIN {X 126.40, Y 83.89, Z 0.00, A 0, B 0, C 0} C_DIS
LIN {X 126.26, Y 84.13, Z 0.00, A 0, B 0, C 0} C_DIS
LIN {X 126.11, Y 84.36, Z 0.00, A 0, B 0, C 0} C_DIS
LIN {X 125.95, Y 84.59, Z 0.00, A 0, B 0, C 0} C_DIS
LIN {X 125.79, Y 84.82, Z 0.00, A 0, B 0, C 0} C_DIS
LIN {X 125.64, Y 85.06, Z 0.00, A 0, B 0, C 0} C_DIS
LIN {X 125.51, Y 85.31, Z 0.00, A 0, B 0, C 0} C_DIS
LIN {X 125.39, Y 85.59, Z 0.00, A 0, B 0, C 0} C_DIS
LIN {X 125.27, Y 85.87, Z 0.00, A 0, B 0, C 0} C_DIS
LIN {X 125.16, Y 86.15, Z 0.00, A 0, B 0, C 0} C_DIS
LIN {X 125.04, Y 86.43, Z 0.00, A 0, B 0, C 0} C_DIS
LIN {X 124.92, Y 86.70, Z 0.00, A 0, B 0, C 0} C_DIS
LIN {X 124.79, Y 86.95, Z 0.00, A 0, B 0, C 0} C_DIS
LIN {X 124.64, Y 87.20, Z 0.00, A 0, B 0, C 0} C_DIS
LIN {X 124.49, Y 87.43, Z 0.00, A 0, B 0, C 0} C_DIS
LIN {X 124.34, Y 87.67, Z 0.00, A 0, B 0, C 0} C_DIS
LIN {X 124.19, Y 87.90, Z 0.00, A 0, B 0, C 0} C_DIS
LIN {X 124.03, Y 88.13, Z 0.00, A 0, B 0, C 0} C_DIS
LIN {X 123.88, Y 88.37, Z 0.00, A 0, B 0, C 0} C_DIS
LIN {X 123.73, Y 88.60, Z 0.00, A 0, B 0, C 0} C_DIS
LIN {X 123.58, Y 88.83, Z 0.00, A 0, B 0, C 0} C_DIS
LIN {X 123.42, Y 89.06, Z 0.00, A 0, B 0, C 0} C_DIS
LIN {X 123.26, Y 89.27, Z 0.00, A 0, B 0, C 0} C_DIS
LIN {X 123.09, Y 89.48, Z 0.00, A 0, B 0, C 0} C_DIS
LIN {X 122.91, Y 89.67, Z 0.00, A 0, B 0, C 0} C_DIS
LIN {X 122.73, Y 89.85, Z 0.00, A 0, B 0, C 0} C_DIS
LIN {X 122.55, Y 90.03, Z 0.00, A 0, B 0, C 0} C_DIS
LIN {X 122.36, Y 90.20, Z 0.00, A 0, B 0, C 0} C_DIS
LIN {X 122.18, Y 90.38, Z 0.00, A 0, B 0, C 0} C_DIS
LIN {X 122.00, Y 90.57, Z 0.00, A 0, B 0, C 0} C_DIS
LIN {X 121.84, Y 90.78, Z 0.00, A 0, B 0, C 0} C_DIS
LIN {X 121.68, Y 91.01, Z 0.00, A 0, B 0, C 0} C_DIS
LIN {X 121.53, Y 91.24, Z 0.00, A 0, B 0, C 0} C_DIS
LIN {X 121.38, Y 91.48, Z 0.00, A 0, B 0, C 0} C_DIS
LIN {X 121.23, Y 91.71, Z 0.00, A 0, B 0, C 0} C_DIS
LIN {X 121.07, Y 91.93, Z 0.00, A 0, B 0, C 0} C_DIS
LIN {X 120.89, Y 92.13, Z 0.00, A 0, B 0, C 0} C_DIS
LIN {X 120.71, Y 92.31, Z 0.00, A 0, B 0, C 0} C_DIS
LIN {X 120.53, Y 92.49, Z 0.00, A 0, B 0, C 0} C_DIS
LIN {X 120.34, Y 92.66, Z 0.00, A 0, B 0, C 0} C_DIS
LIN {X 120.15, Y 92.81, Z 0.00, A 0, B 0, C 0} C_DIS
LIN {X 119.96, Y 92.95, Z 0.00, A 0, B 0, C 0} C_DIS
LIN {X 119.76, Y 93.09, Z 0.00, A 0, B 0, C 0} C_DIS
LIN {X 119.57, Y 93.24, Z 0.00, A 0, B 0, C 0} C_DIS
LIN {X 119.38, Y 93.41, Z 0.00, A 0, B 0, C 0} C_DIS
LIN {X 119.20, Y 93.59, Z 0.00, A 0, B 0, C 0} C_DIS
LIN {X 119.02, Y 93.77, Z 0.00, A 0, B 0, C 0} C_DIS
LIN {X 118.84, Y 93.96, Z 0.00, A 0, B 0, C 0} C_DIS
LIN {X 118.66, Y 94.16, Z 0.00, A 0, B 0, C 0} C_DIS
LIN {X 118.48, Y 94.34, Z 0.00, A 0, B 0, C 0} C_DIS
LIN {X 118.30, Y 94.52, Z 0.00, A 0, B 0, C 0} C_DIS
LIN {X 118.11, Y 94.68, Z 0.00, A 0, B 0, C 0} C_DIS
LIN {X 117.92, Y 94.82, Z 0.00, A 0, B 0, C 0} C_DIS
LIN {X 117.72, Y 94.95, Z 0.00, A 0, B 0, C 0} C_DIS
LIN {X 117.52, Y 95.09, Z 0.00, A 0, B 0, C 0} C_DIS
LIN {X 117.33, Y 95.25, Z 0.00, A 0, B 0, C 0} C_DIS
LIN {X 117.15, Y 95.41, Z 0.00, A 0, B 0, C 0} C_DIS
LIN {X 116.95, Y 95.55, Z 0.00, A 0, B 0, C 0} C_DIS
LIN {X 116.75, Y 95.68, Z 0.00, A 0, B 0, C 0} C_DIS
LIN {X 116.55, Y 95.82, Z 0.00, A 0, B 0, C 0} C_DIS
LIN {X 116.37, Y 95.98, Z 0.00, A 0, B 0, C 0} C_DIS
LIN {X 116.18, Y 96.14, Z 0.00, A 0, B 0, C 0} C_DIS
LIN {X 115.97, Y 96.26, Z 0.00, A 0, B 0, C 0} C_DIS
LIN {X 115.78, Y 96.39, Z 0.00, A 0, B 0, C 0} C_DIS
LIN {X 115.61, Y 96.61, Z 0.00, A 0, B 0, C 0} C_DIS
LIN {X 115.46, Y 96.85, Z 0.00, A 0, B 0, C 0} C_DIS
LIN {X 115.31, Y 97.08, Z 0.00, A 0, B 0, C 0} C_DIS
LIN {X 115.16, Y 97.31, Z 0.00, A 0, B 0, C 0} C_DIS
LIN {X 115.04, Y 97.58, Z 0.00, A 0, B 0, C 0} C_DIS
LIN {X 114.95, Y 97.88, Z 0.00, A 0, B 0, C 0} C_DIS
LIN {X 114.89, Y 98.20, Z 0.00, A 0, B 0, C 0} C_DIS
LIN {X 114.84, Y 98.52, Z 0.00, A 0, B 0, C 0} C_DIS
LIN {X 114.80, Y 98.85, Z 0.00, A 0, B 0, C 0} C_DIS
LIN {X 114.77, Y 99.17, Z 0.00, A 0, B 0, C 0} C_DIS
LIN {X 114.75, Y 99.49, Z 0.00, A 0, B 0, C 0} C_DIS
LIN {X 114.74, Y 99.82, Z 0.00, A 0, B 0, C 0} C_DIS
LIN {X 114.73, Y 100.14, Z 0.00, A 0, B 0, C 0} C_DIS
LIN {X 114.73, Y 100.47, Z 0.00, A 0, B 0, C 0} C_DIS
LIN {X 114.72, Y 100.80, Z 0.00, A 0, B 0, C 0} C_DIS
LIN {X 114.72, Y 101.13, Z 0.00, A 0, B 0, C 0} C_DIS
LIN {X 114.73, Y 101.45, Z 0.00, A 0, B 0, C 0} C_DIS
LIN {X 114.73, Y 101.78, Z 0.00, A 0, B 0, C 0} C_DIS
LIN {X 114.73, Y 102.11, Z 0.00, A 0, B 0, C 0} C_DIS
LIN {X 114.74, Y 102.44, Z 0.00, A 0, B 0, C 0} C_DIS
LIN {X 114.74, Y 102.77, Z 0.00, A 0, B 0, C 0} C_DIS
LIN {X 114.74, Y 103.10, Z 0.00, A 0, B 0, C 0} C_DIS
LIN {X 114.74, Y 103.42, Z 0.00, A 0, B 0, C 0} C_DIS
LIN {X 114.74, Y 103.75, Z 0.00, A 0, B 0, C 0} C_DIS
LIN {X 114.74, Y 104.08, Z 0.00, A 0, B 0, C 0} C_DIS
LIN {X 114.73, Y 104.40, Z 0.00, A 0, B 0, C 0} C_DIS
LIN {X 114.73, Y 104.73, Z 0.00, A 0, B 0, C 0} C_DIS
LIN {X 114.73, Y 105.06, Z 0.00, A 0, B 0, C 0} C_DIS
LIN {X 114.73, Y 105.39, Z 0.00, A 0, B 0, C 0} C_DIS
LIN {X 114.73, Y 105.72, Z 0.00, A 0, B 0, C 0} C_DIS
LIN {X 114.73, Y 106.04, Z 0.00, A 0, B 0, C 0} C_DIS
LIN {X 114.74, Y 106.37, Z 0.00, A 0, B 0, C 0} C_DIS
LIN {X 114.74, Y 106.70, Z 0.00, A 0, B 0, C 0} C_DIS
LIN {X 114.74, Y 107.03, Z 0.00, A 0, B 0, C 0} C_DIS
LIN {X 114.73, Y 107.35, Z 0.00, A 0, B 0, C 0} C_DIS
LIN {X 114.72, Y 107.68, Z 0.00, A 0, B 0, C 0} C_DIS
LIN {X 114.69, Y 108.01, Z 0.00, A 0, B 0, C 0} C_DIS
LIN {X 114.65, Y 108.33, Z 0.00, A 0, B 0, C 0} C_DIS
LIN {X 114.58, Y 108.64, Z 0.00, A 0, B 0, C 0} C_DIS
LIN {X 114.48, Y 108.93, Z 0.00, A 0, B 0, C 0} C_DIS
LIN {X 114.34, Y 109.17, Z 0.00, A 0, B 0, C 0} C_DIS
LIN {X 114.17, Y 109.38, Z 0.00, A 0, B 0, C 0} C_DIS
LIN {X 113.99, Y 109.56, Z 0.00, A 0, B 0, C 0} C_DIS
LIN {X 113.80, Y 109.72, Z 0.00, A 0, B 0, C 0} C_DIS
LIN {X 113.60, Y 109.86, Z 0.00, A 0, B 0, C 0} C_DIS
LIN {X 113.41, Y 110.00, Z 0.00, A 0, B 0, C 0} C_DIS
LIN {X 113.21, Y 110.14, Z 0.00, A 0, B 0, C 0} C_DIS
LIN {X 113.02, Y 110.30, Z 0.00, A 0, B 0, C 0} C_DIS
LIN {X 112.84, Y 110.47, Z 0.00, A 0, B 0, C 0} C_DIS
LIN {X 112.65, Y 110.65, Z 0.00, A 0, B 0, C 0} C_DIS
LIN {X 112.48, Y 110.84, Z 0.00, A 0, B 0, C 0} C_DIS
LIN {X 112.30, Y 111.03, Z 0.00, A 0, B 0, C 0} C_DIS
LIN {X 112.12, Y 111.22, Z 0.00, A 0, B 0, C 0} C_DIS
LIN {X 111.94, Y 111.40, Z 0.00, A 0, B 0, C 0} C_DIS
LIN {X 111.76, Y 111.58, Z 0.00, A 0, B 0, C 0} C_DIS
LIN {X 111.57, Y 111.73, Z 0.00, A 0, B 0, C 0} C_DIS
LIN {X 111.37, Y 111.87, Z 0.00, A 0, B 0, C 0} C_DIS
LIN {X 111.17, Y 112.00, Z 0.00, A 0, B 0, C 0} C_DIS
LIN {X 110.98, Y 112.15, Z 0.00, A 0, B 0, C 0} C_DIS
LIN {X 110.79, Y 112.32, Z 0.00, A 0, B 0, C 0} C_DIS
LIN {X 110.60, Y 112.47, Z 0.00, A 0, B 0, C 0} C_DIS
LIN {X 110.40, Y 112.59, Z 0.00, A 0, B 0, C 0} C_DIS
LIN {X 110.20, Y 112.73, Z 0.00, A 0, B 0, C 0} C_DIS
LIN {X 110.01, Y 112.89, Z 0.00, A 0, B 0, C 0} C_DIS
LIN {X 109.83, Y 113.06, Z 0.00, A 0, B 0, C 0} C_DIS
LIN {X 109.65, Y 113.24, Z 0.00, A 0, B 0, C 0} C_DIS
LIN {X 109.47, Y 113.43, Z 0.00, A 0, B 0, C 0} C_DIS
LIN {X 109.29, Y 113.61, Z 0.00, A 0, B 0, C 0} C_DIS
LIN {X 109.11, Y 113.80, Z 0.00, A 0, B 0, C 0} C_DIS
LIN {X 108.93, Y 113.99, Z 0.00, A 0, B 0, C 0} C_DIS
LIN {X 108.75, Y 114.16, Z 0.00, A 0, B 0, C 0} C_DIS
LIN {X 108.56, Y 114.33, Z 0.00, A 0, B 0, C 0} C_DIS
LIN {X 108.36, Y 114.47, Z 0.00, A 0, B 0, C 0} C_DIS
LIN {X 108.17, Y 114.61, Z 0.00, A 0, B 0, C 0} C_DIS
LIN {X 107.97, Y 114.75, Z 0.00, A 0, B 0, C 0} C_DIS
LIN {X 107.78, Y 114.91, Z 0.00, A 0, B 0, C 0} C_DIS
LIN {X 107.60, Y 115.08, Z 0.00, A 0, B 0, C 0} C_DIS
LIN {X 107.42, Y 115.26, Z 0.00, A 0, B 0, C 0} C_DIS
LIN {X 107.24, Y 115.45, Z 0.00, A 0, B 0, C 0} C_DIS
LIN {X 107.06, Y 115.64, Z 0.00, A 0, B 0, C 0} C_DIS
LIN {X 106.88, Y 115.83, Z 0.00, A 0, B 0, C 0} C_DIS
LIN {X 106.70, Y 116.01, Z 0.00, A 0, B 0, C 0} C_DIS
LIN {X 106.52, Y 116.18, Z 0.00, A 0, B 0, C 0} C_DIS
LIN {X 106.33, Y 116.34, Z 0.00, A 0, B 0, C 0} C_DIS
LIN {X 106.13, Y 116.48, Z 0.00, A 0, B 0, C 0} C_DIS
LIN {X 105.93, Y 116.61, Z 0.00, A 0, B 0, C 0} C_DIS
LIN {X 105.74, Y 116.75, Z 0.00, A 0, B 0, C 0} C_DIS
LIN {X 105.55, Y 116.92, Z 0.00, A 0, B 0, C 0} C_DIS
LIN {X 105.36, Y 117.07, Z 0.00, A 0, B 0, C 0} C_DIS
LIN {X 105.16, Y 117.20, Z 0.00, A 0, B 0, C 0} C_DIS
LIN {X 104.96, Y 117.33, Z 0.00, A 0, B 0, C 0} C_DIS
LIN {X 104.77, Y 117.49, Z 0.00, A 0, B 0, C 0} C_DIS
LIN {X 104.59, Y 117.67, Z 0.00, A 0, B 0, C 0} C_DIS
LIN {X 104.41, Y 117.86, Z 0.00, A 0, B 0, C 0} C_DIS
LIN {X 104.23, Y 118.05, Z 0.00, A 0, B 0, C 0} C_DIS
LIN {X 104.05, Y 118.23, Z 0.00, A 0, B 0, C 0} C_DIS
LIN {X 103.87, Y 118.40, Z 0.00, A 0, B 0, C 0} C_DIS
LIN {X 103.69, Y 118.58, Z 0.00, A 0, B 0, C 0} C_DIS
LIN {X 103.51, Y 118.77, Z 0.00, A 0, B 0, C 0} C_DIS
LIN {X 103.32, Y 118.95, Z 0.00, A 0, B 0, C 0} C_DIS
LIN {X 103.12, Y 119.08, Z 0.00, A 0, B 0, C 0} C_DIS
LIN {X 102.92, Y 119.20, Z 0.00, A 0, B 0, C 0} C_DIS
LIN {X 102.73, Y 119.35, Z 0.00, A 0, B 0, C 0} C_DIS
LIN {X 102.54, Y 119.51, Z 0.00, A 0, B 0, C 0} C_DIS
LIN {X 102.36, Y 119.69, Z 0.00, A 0, B 0, C 0} C_DIS
LIN {X 102.18, Y 119.87, Z 0.00, A 0, B 0, C 0} C_DIS
LIN {X 102.00, Y 120.06, Z 0.00, A 0, B 0, C 0} C_DIS
LIN {X 101.82, Y 120.25, Z 0.00, A 0, B 0, C 0} C_DIS
LIN {X 101.64, Y 120.43, Z 0.00, A 0, B 0, C 0} C_DIS
LIN {X 101.46, Y 120.61, Z 0.00, A 0, B 0, C 0} C_DIS
LIN {X 101.28, Y 120.78, Z 0.00, A 0, B 0, C 0} C_DIS
LIN {X 101.09, Y 120.94, Z 0.00, A 0, B 0, C 0} C_DIS
LIN {X 100.89, Y 121.09, Z 0.00, A 0, B 0, C 0} C_DIS
LIN {X 100.69, Y 121.21, Z 0.00, A 0, B 0, C 0} C_DIS
LIN {X 100.50, Y 121.36, Z 0.00, A 0, B 0, C 0} C_DIS
LIN {X 100.31, Y 121.52, Z 0.00, A 0, B 0, C 0} C_DIS
LIN {X 100.12, Y 121.67, Z 0.00, A 0, B 0, C 0} C_DIS
LIN {X 99.92, Y 121.81, Z 0.00, A 0, B 0, C 0} C_DIS
LIN {X 99.72, Y 121.95, Z 0.00, A 0, B 0, C 0} C_DIS
LIN {X 99.53, Y 122.10, Z 0.00, A 0, B 0, C 0} C_DIS
LIN {X 99.35, Y 122.27, Z 0.00, A 0, B 0, C 0} C_DIS
LIN {X 99.17, Y 122.45, Z 0.00, A 0, B 0, C 0} C_DIS
LIN {X 98.99, Y 122.64, Z 0.00, A 0, B 0, C 0} C_DIS
LIN {X 98.81, Y 122.84, Z 0.00, A 0, B 0, C 0} C_DIS
LIN {X 98.63, Y 123.03, Z 0.00, A 0, B 0, C 0} C_DIS
LIN {X 98.45, Y 123.21, Z 0.00, A 0, B 0, C 0} C_DIS
LIN {X 98.27, Y 123.37, Z 0.00, A 0, B 0, C 0} C_DIS
LIN {X 98.07, Y 123.53, Z 0.00, A 0, B 0, C 0} C_DIS
LIN {X 97.88, Y 123.67, Z 0.00, A 0, B 0, C 0} C_DIS
LIN {X 97.69, Y 123.82, Z 0.00, A 0, B 0, C 0} C_DIS
LIN {X 97.49, Y 123.96, Z 0.00, A 0, B 0, C 0} C_DIS
LIN {X 97.30, Y 124.12, Z 0.00, A 0, B 0, C 0} C_DIS
LIN {X 97.12, Y 124.29, Z 0.00, A 0, B 0, C 0} C_DIS
LIN {X 96.94, Y 124.47, Z 0.00, A 0, B 0, C 0} C_DIS
LIN {X 96.76, Y 124.66, Z 0.00, A 0, B 0, C 0} C_DIS
LIN {X 96.58, Y 124.86, Z 0.00, A 0, B 0, C 0} C_DIS
LIN {X 96.40, Y 125.05, Z 0.00, A 0, B 0, C 0} C_DIS
LIN {X 96.22, Y 125.23, Z 0.00, A 0, B 0, C 0} C_DIS
LIN {X 96.04, Y 125.39, Z 0.00, A 0, B 0, C 0} C_DIS
LIN {X 95.84, Y 125.54, Z 0.00, A 0, B 0, C 0} C_DIS
LIN {X 95.65, Y 125.68, Z 0.00, A 0, B 0, C 0} C_DIS
LIN {X 95.45, Y 125.81, Z 0.00, A 0, B 0, C 0} C_DIS
LIN {X 95.26, Y 125.97, Z 0.00, A 0, B 0, C 0} C_DIS
LIN {X 95.07, Y 126.14, Z 0.00, A 0, B 0, C 0} C_DIS
LIN {X 94.87, Y 126.27, Z 0.00, A 0, B 0, C 0} C_DIS
LIN {X 94.67, Y 126.40, Z 0.00, A 0, B 0, C 0} C_DIS
LIN {X 94.48, Y 126.55, Z 0.00, A 0, B 0, C 0} C_DIS
LIN {X 94.29, Y 126.71, Z 0.00, A 0, B 0, C 0} C_DIS
LIN {X 94.11, Y 126.88, Z 0.00, A 0, B 0, C 0} C_DIS
LIN {X 93.93, Y 127.07, Z 0.00, A 0, B 0, C 0} C_DIS
LIN {X 93.75, Y 127.25, Z 0.00, A 0, B 0, C 0} C_DIS
LIN {X 93.57, Y 127.44, Z 0.00, A 0, B 0, C 0} C_DIS
LIN {X 93.39, Y 127.63, Z 0.00, A 0, B 0, C 0} C_DIS
LIN {X 93.21, Y 127.81, Z 0.00, A 0, B 0, C 0} C_DIS
LIN {X 93.03, Y 127.98, Z 0.00, A 0, B 0, C 0} C_DIS
LIN {X 92.84, Y 128.14, Z 0.00, A 0, B 0, C 0} C_DIS
LIN {X 92.64, Y 128.28, Z 0.00, A 0, B 0, C 0} C_DIS
LIN {X 92.44, Y 128.42, Z 0.00, A 0, B 0, C 0} C_DIS
LIN {X 92.25, Y 128.56, Z 0.00, A 0, B 0, C 0} C_DIS
LIN {X 92.06, Y 128.73, Z 0.00, A 0, B 0, C 0} C_DIS
LIN {X 91.88, Y 128.90, Z 0.00, A 0, B 0, C 0} C_DIS
LIN {X 91.70, Y 129.08, Z 0.00, A 0, B 0, C 0} C_DIS
LIN {X 91.52, Y 129.27, Z 0.00, A 0, B 0, C 0} C_DIS
LIN {X 91.34, Y 129.46, Z 0.00, A 0, B 0, C 0} C_DIS
LIN {X 91.16, Y 129.65, Z 0.00, A 0, B 0, C 0} C_DIS
LIN {X 90.98, Y 129.83, Z 0.00, A 0, B 0, C 0} C_DIS
LIN {X 90.80, Y 130.00, Z 0.00, A 0, B 0, C 0} C_DIS
LIN {X 90.61, Y 130.15, Z 0.00, A 0, B 0, C 0} C_DIS
LIN {X 90.41, Y 130.29, Z 0.00, A 0, B 0, C 0} C_DIS
LIN {X 90.21, Y 130.41, Z 0.00, A 0, B 0, C 0} C_DIS
LIN {X 90.02, Y 130.57, Z 0.00, A 0, B 0, C 0} C_DIS
LIN {X 89.83, Y 130.75, Z 0.00, A 0, B 0, C 0} C_DIS
LIN {X 89.63, Y 130.88, Z 0.00, A 0, B 0, C 0} C_DIS
LIN {X 89.43, Y 131.01, Z 0.00, A 0, B 0, C 0} C_DIS
LIN {X 89.24, Y 131.15, Z 0.00, A 0, B 0, C 0} C_DIS
LIN {X 89.05, Y 131.31, Z 0.00, A 0, B 0, C 0} C_DIS
LIN {X 88.87, Y 131.49, Z 0.00, A 0, B 0, C 0} C_DIS
LIN {X 88.69, Y 131.67, Z 0.00, A 0, B 0, C 0} C_DIS
LIN {X 88.51, Y 131.86, Z 0.00, A 0, B 0, C 0} C_DIS
LIN {X 88.33, Y 132.05, Z 0.00, A 0, B 0, C 0} C_DIS
LIN {X 88.15, Y 132.24, Z 0.00, A 0, B 0, C 0} C_DIS
LIN {X 87.97, Y 132.42, Z 0.00, A 0, B 0, C 0} C_DIS
LIN {X 87.79, Y 132.59, Z 0.00, A 0, B 0, C 0} C_DIS
LIN {X 87.60, Y 132.74, Z 0.00, A 0, B 0, C 0} C_DIS
LIN {X 87.40, Y 132.88, Z 0.00, A 0, B 0, C 0} C_DIS
LIN {X 87.20, Y 133.01, Z 0.00, A 0, B 0, C 0} C_DIS
LIN {X 87.01, Y 133.17, Z 0.00, A 0, B 0, C 0} C_DIS
LIN {X 86.83, Y 133.34, Z 0.00, A 0, B 0, C 0} C_DIS
LIN {X 86.64, Y 133.52, Z 0.00, A 0, B 0, C 0} C_DIS
LIN {X 86.46, Y 133.70, Z 0.00, A 0, B 0, C 0} C_DIS
LIN {X 86.28, Y 133.88, Z 0.00, A 0, B 0, C 0} C_DIS
LIN {X 86.10, Y 134.07, Z 0.00, A 0, B 0, C 0} C_DIS
LIN {X 85.92, Y 134.26, Z 0.00, A 0, B 0, C 0} C_DIS
LIN {X 85.74, Y 134.44, Z 0.00, A 0, B 0, C 0} C_DIS
LIN {X 85.56, Y 134.61, Z 0.00, A 0, B 0, C 0} C_DIS
LIN {X 85.37, Y 134.76, Z 0.00, A 0, B 0, C 0} C_DIS
LIN {X 85.17, Y 134.89, Z 0.00, A 0, B 0, C 0} C_DIS
LIN {X 84.97, Y 135.02, Z 0.00, A 0, B 0, C 0} C_DIS
LIN {X 84.78, Y 135.18, Z 0.00, A 0, B 0, C 0} C_DIS
LIN {X 84.59, Y 135.35, Z 0.00, A 0, B 0, C 0} C_DIS
LIN {X 84.39, Y 135.48, Z 0.00, A 0, B 0, C 0} C_DIS
LIN {X 84.19, Y 135.61, Z 0.00, A 0, B 0, C 0} C_DIS
LIN {X 84.00, Y 135.76, Z 0.00, A 0, B 0, C 0} C_DIS
LIN {X 83.81, Y 135.92, Z 0.00, A 0, B 0, C 0} C_DIS
LIN {X 83.63, Y 136.10, Z 0.00, A 0, B 0, C 0} C_DIS
LIN {X 83.45, Y 136.29, Z 0.00, A 0, B 0, C 0} C_DIS
LIN {X 83.27, Y 136.48, Z 0.00, A 0, B 0, C 0} C_DIS
LIN {X 83.10, Y 136.67, Z 0.00, A 0, B 0, C 0} C_DIS
LIN {X 82.92, Y 136.85, Z 0.00, A 0, B 0, C 0} C_DIS
LIN {X 82.73, Y 137.03, Z 0.00, A 0, B 0, C 0} C_DIS
LIN {X 82.54, Y 137.19, Z 0.00, A 0, B 0, C 0} C_DIS
LIN {X 82.35, Y 137.34, Z 0.00, A 0, B 0, C 0} C_DIS
LIN {X 82.16, Y 137.49, Z 0.00, A 0, B 0, C 0} C_DIS
LIN {X 81.97, Y 137.63, Z 0.00, A 0, B 0, C 0} C_DIS
LIN {X 81.77, Y 137.78, Z 0.00, A 0, B 0, C 0} C_DIS
LIN {X 81.58, Y 137.94, Z 0.00, A 0, B 0, C 0} C_DIS
LIN {X 81.40, Y 138.12, Z 0.00, A 0, B 0, C 0} C_DIS
LIN {X 81.22, Y 138.30, Z 0.00, A 0, B 0, C 0} C_DIS
LIN {X 81.04, Y 138.49, Z 0.00, A 0, B 0, C 0} C_DIS
LIN {X 80.86, Y 138.68, Z 0.00, A 0, B 0, C 0} C_DIS
LIN {X 80.69, Y 138.87, Z 0.00, A 0, B 0, C 0} C_DIS
LIN {X 80.50, Y 139.05, Z 0.00, A 0, B 0, C 0} C_DIS
LIN {X 80.32, Y 139.21, Z 0.00, A 0, B 0, C 0} C_DIS
LIN {X 80.12, Y 139.36, Z 0.00, A 0, B 0, C 0} C_DIS
LIN {X 79.93, Y 139.49, Z 0.00, A 0, B 0, C 0} C_DIS
LIN {X 79.72, Y 139.62, Z 0.00, A 0, B 0, C 0} C_DIS
LIN {X 79.54, Y 139.79, Z 0.00, A 0, B 0, C 0} C_DIS
LIN {X 79.35, Y 139.95, Z 0.00, A 0, B 0, C 0} C_DIS
LIN {X 79.15, Y 140.08, Z 0.00, A 0, B 0, C 0} C_DIS
LIN {X 78.95, Y 140.21, Z 0.00, A 0, B 0, C 0} C_DIS
LIN {X 78.76, Y 140.36, Z 0.00, A 0, B 0, C 0} C_DIS
LIN {X 78.57, Y 140.53, Z 0.00, A 0, B 0, C 0} C_DIS
LIN {X 78.39, Y 140.71, Z 0.00, A 0, B 0, C 0} C_DIS
LIN {X 78.21, Y 140.89, Z 0.00, A 0, B 0, C 0} C_DIS
LIN {X 78.03, Y 141.08, Z 0.00, A 0, B 0, C 0} C_DIS
LIN {X 77.86, Y 141.27, Z 0.00, A 0, B 0, C 0} C_DIS
LIN {X 77.68, Y 141.46, Z 0.00, A 0, B 0, C 0} C_DIS
LIN {X 77.49, Y 141.64, Z 0.00, A 0, B 0, C 0} C_DIS
LIN {X 77.31, Y 141.80, Z 0.00, A 0, B 0, C 0} C_DIS
LIN {X 77.11, Y 141.94, Z 0.00, A 0, B 0, C 0} C_DIS
LIN {X 76.92, Y 142.09, Z 0.00, A 0, B 0, C 0} C_DIS
LIN {X 76.72, Y 142.23, Z 0.00, A 0, B 0, C 0} C_DIS
LIN {X 76.53, Y 142.39, Z 0.00, A 0, B 0, C 0} C_DIS
LIN {X 76.34, Y 142.55, Z 0.00, A 0, B 0, C 0} C_DIS
LIN {X 76.16, Y 142.73, Z 0.00, A 0, B 0, C 0} C_DIS
LIN {X 75.98, Y 142.91, Z 0.00, A 0, B 0, C 0} C_DIS
LIN {X 75.80, Y 143.10, Z 0.00, A 0, B 0, C 0} C_DIS
LIN {X 75.63, Y 143.29, Z 0.00, A 0, B 0, C 0} C_DIS
LIN {X 75.45, Y 143.48, Z 0.00, A 0, B 0, C 0} C_DIS
LIN {X 75.26, Y 143.65, Z 0.00, A 0, B 0, C 0} C_DIS
LIN {X 75.08, Y 143.81, Z 0.00, A 0, B 0, C 0} C_DIS
LIN {X 74.88, Y 143.96, Z 0.00, A 0, B 0, C 0} C_DIS
LIN {X 74.68, Y 144.10, Z 0.00, A 0, B 0, C 0} C_DIS
LIN {X 74.49, Y 144.24, Z 0.00, A 0, B 0, C 0} C_DIS
LIN {X 74.30, Y 144.40, Z 0.00, A 0, B 0, C 0} C_DIS
LIN {X 74.11, Y 144.57, Z 0.00, A 0, B 0, C 0} C_DIS
LIN {X 73.93, Y 144.75, Z 0.00, A 0, B 0, C 0} C_DIS
LIN {X 73.75, Y 144.94, Z 0.00, A 0, B 0, C 0} C_DIS
LIN {X 73.58, Y 145.13, Z 0.00, A 0, B 0, C 0} C_DIS
LIN {X 73.40, Y 145.31, Z 0.00, A 0, B 0, C 0} C_DIS
LIN {X 73.22, Y 145.50, Z 0.00, A 0, B 0, C 0} C_DIS
LIN {X 73.03, Y 145.67, Z 0.00, A 0, B 0, C 0} C_DIS
LIN {X 72.84, Y 145.83, Z 0.00, A 0, B 0, C 0} C_DIS
LIN {X 72.65, Y 145.97, Z 0.00, A 0, B 0, C 0} C_DIS
LIN {X 72.45, Y 146.11, Z 0.00, A 0, B 0, C 0} C_DIS
LIN {X 72.26, Y 146.25, Z 0.00, A 0, B 0, C 0} C_DIS
LIN {X 72.07, Y 146.41, Z 0.00, A 0, B 0, C 0} C_DIS
LIN {X 71.88, Y 146.59, Z 0.00, A 0, B 0, C 0} C_DIS
LIN {X 71.70, Y 146.77, Z 0.00, A 0, B 0, C 0} C_DIS
LIN {X 71.53, Y 146.96, Z 0.00, A 0, B 0, C 0} C_DIS
LIN {X 71.35, Y 147.15, Z 0.00, A 0, B 0, C 0} C_DIS
LIN {X 71.17, Y 147.34, Z 0.00, A 0, B 0, C 0} C_DIS
LIN {X 70.99, Y 147.52, Z 0.00, A 0, B 0, C 0} C_DIS
LIN {X 70.80, Y 147.69, Z 0.00, A 0, B 0, C 0} C_DIS
LIN {X 70.61, Y 147.84, Z 0.00, A 0, B 0, C 0} C_DIS
LIN {X 70.41, Y 147.97, Z 0.00, A 0, B 0, C 0} C_DIS
LIN {X 70.22, Y 148.11, Z 0.00, A 0, B 0, C 0} C_DIS
LIN {X 70.03, Y 148.26, Z 0.00, A 0, B 0, C 0} C_DIS
LIN {X 69.84, Y 148.43, Z 0.00, A 0, B 0, C 0} C_DIS
LIN {X 69.66, Y 148.61, Z 0.00, A 0, B 0, C 0} C_DIS
LIN {X 69.48, Y 148.80, Z 0.00, A 0, B 0, C 0} C_DIS
LIN {X 69.30, Y 148.98, Z 0.00, A 0, B 0, C 0} C_DIS
LIN {X 69.12, Y 149.17, Z 0.00, A 0, B 0, C 0} C_DIS
LIN {X 68.94, Y 149.36, Z 0.00, A 0, B 0, C 0} C_DIS
LIN {X 68.76, Y 149.53, Z 0.00, A 0, B 0, C 0} C_DIS
LIN {X 68.57, Y 149.70, Z 0.00, A 0, B 0, C 0} C_DIS
LIN {X 68.38, Y 149.85, Z 0.00, A 0, B 0, C 0} C_DIS
LIN {X 68.18, Y 149.99, Z 0.00, A 0, B 0, C 0} C_DIS
LIN {X 67.98, Y 150.12, Z 0.00, A 0, B 0, C 0} C_DIS
LIN {X 67.79, Y 150.27, Z 0.00, A 0, B 0, C 0} C_DIS
LIN {X 67.61, Y 150.44, Z 0.00, A 0, B 0, C 0} C_DIS
LIN {X 67.43, Y 150.63, Z 0.00, A 0, B 0, C 0} C_DIS
LIN {X 67.25, Y 150.82, Z 0.00, A 0, B 0, C 0} C_DIS
LIN {X 67.07, Y 151.01, Z 0.00, A 0, B 0, C 0} C_DIS
LIN {X 66.89, Y 151.20, Z 0.00, A 0, B 0, C 0} C_DIS
LIN {X 66.71, Y 151.38, Z 0.00, A 0, B 0, C 0} C_DIS
LIN {X 66.53, Y 151.55, Z 0.00, A 0, B 0, C 0} C_DIS
LIN {X 66.34, Y 151.71, Z 0.00, A 0, B 0, C 0} C_DIS
LIN {X 66.14, Y 151.85, Z 0.00, A 0, B 0, C 0} C_DIS
LIN {X 65.94, Y 151.98, Z 0.00, A 0, B 0, C 0} C_DIS
LIN {X 65.75, Y 152.13, Z 0.00, A 0, B 0, C 0} C_DIS
LIN {X 65.57, Y 152.30, Z 0.00, A 0, B 0, C 0} C_DIS
LIN {X 65.38, Y 152.48, Z 0.00, A 0, B 0, C 0} C_DIS
LIN {X 65.20, Y 152.65, Z 0.00, A 0, B 0, C 0} C_DIS
LIN {X 65.02, Y 152.84, Z 0.00, A 0, B 0, C 0} C_DIS
LIN {X 64.84, Y 153.03, Z 0.00, A 0, B 0, C 0} C_DIS
LIN {X 64.66, Y 153.22, Z 0.00, A 0, B 0, C 0} C_DIS
LIN {X 64.48, Y 153.40, Z 0.00, A 0, B 0, C 0} C_DIS
LIN {X 64.30, Y 153.57, Z 0.00, A 0, B 0, C 0} C_DIS
LIN {X 64.11, Y 153.72, Z 0.00, A 0, B 0, C 0} C_DIS
LIN {X 63.91, Y 153.86, Z 0.00, A 0, B 0, C 0} C_DIS
LIN {X 63.71, Y 154.00, Z 0.00, A 0, B 0, C 0} C_DIS
LIN {X 63.52, Y 154.15, Z 0.00, A 0, B 0, C 0} C_DIS
LIN {X 63.33, Y 154.31, Z 0.00, A 0, B 0, C 0} C_DIS
LIN {X 63.15, Y 154.49, Z 0.00, A 0, B 0, C 0} C_DIS
LIN {X 62.97, Y 154.68, Z 0.00, A 0, B 0, C 0} C_DIS
LIN {X 62.80, Y 154.87, Z 0.00, A 0, B 0, C 0} C_DIS
LIN {X 62.61, Y 155.05, Z 0.00, A 0, B 0, C 0} C_DIS
LIN {X 62.43, Y 155.23, Z 0.00, A 0, B 0, C 0} C_DIS
LIN {X 62.25, Y 155.41, Z 0.00, A 0, B 0, C 0} C_DIS
LIN {X 62.07, Y 155.60, Z 0.00, A 0, B 0, C 0} C_DIS
LIN {X 61.88, Y 155.74, Z 0.00, A 0, B 0, C 0} C_DIS
LIN {X 61.67, Y 155.86, Z 0.00, A 0, B 0, C 0} C_DIS
LIN {X 61.48, Y 156.00, Z 0.00, A 0, B 0, C 0} C_DIS
LIN {X 61.29, Y 156.16, Z 0.00, A 0, B 0, C 0} C_DIS
LIN {X 61.11, Y 156.33, Z 0.00, A 0, B 0, C 0} C_DIS
LIN {X 60.93, Y 156.52, Z 0.00, A 0, B 0, C 0} C_DIS
LIN {X 60.75, Y 156.70, Z 0.00, A 0, B 0, C 0} C_DIS
LIN {X 60.57, Y 156.89, Z 0.00, A 0, B 0, C 0} C_DIS
LIN {X 60.38, Y 157.07, Z 0.00, A 0, B 0, C 0} C_DIS
LIN {X 60.20, Y 157.25, Z 0.00, A 0, B 0, C 0} C_DIS
LIN {X 60.02, Y 157.43, Z 0.00, A 0, B 0, C 0} C_DIS
LIN {X 59.83, Y 157.59, Z 0.00, A 0, B 0, C 0} C_DIS
LIN {X 59.64, Y 157.74, Z 0.00, A 0, B 0, C 0} C_DIS
LIN {X 59.45, Y 157.88, Z 0.00, A 0, B 0, C 0} C_DIS
LIN {X 59.25, Y 158.02, Z 0.00, A 0, B 0, C 0} C_DIS
LIN {X 59.06, Y 158.18, Z 0.00, A 0, B 0, C 0} C_DIS
LIN {X 58.87, Y 158.35, Z 0.00, A 0, B 0, C 0} C_DIS
LIN {X 58.69, Y 158.53, Z 0.00, A 0, B 0, C 0} C_DIS
LIN {X 58.51, Y 158.71, Z 0.00, A 0, B 0, C 0} C_DIS
LIN {X 58.33, Y 158.90, Z 0.00, A 0, B 0, C 0} C_DIS
LIN {X 58.16, Y 159.09, Z 0.00, A 0, B 0, C 0} C_DIS
LIN {X 57.98, Y 159.28, Z 0.00, A 0, B 0, C 0} C_DIS
LIN {X 57.80, Y 159.46, Z 0.00, A 0, B 0, C 0} C_DIS
LIN {X 57.61, Y 159.64, Z 0.00, A 0, B 0, C 0} C_DIS
LIN {X 57.43, Y 159.81, Z 0.00, A 0, B 0, C 0} C_DIS
LIN {X 57.25, Y 159.99, Z 0.00, A 0, B 0, C 0} C_DIS
LIN {X 57.07, Y 160.17, Z 0.00, A 0, B 0, C 0} C_DIS
LIN {X 56.89, Y 160.36, Z 0.00, A 0, B 0, C 0} C_DIS
LIN {X 56.71, Y 160.55, Z 0.00, A 0, B 0, C 0} C_DIS
LIN {X 56.53, Y 160.73, Z 0.00, A 0, B 0, C 0} C_DIS
LIN {X 56.34, Y 160.90, Z 0.00, A 0, B 0, C 0} C_DIS
LIN {X 56.14, Y 161.03, Z 0.00, A 0, B 0, C 0} C_DIS
LIN {X 55.94, Y 161.15, Z 0.00, A 0, B 0, C 0} C_DIS
LIN {X 55.75, Y 161.29, Z 0.00, A 0, B 0, C 0} C_DIS
LIN {X 55.56, Y 161.47, Z 0.00, A 0, B 0, C 0} C_DIS
LIN {X 55.38, Y 161.65, Z 0.00, A 0, B 0, C 0} C_DIS
LIN {X 55.20, Y 161.84, Z 0.00, A 0, B 0, C 0} C_DIS
LIN {X 55.02, Y 162.02, Z 0.00, A 0, B 0, C 0} C_DIS
LIN {X 54.84, Y 162.20, Z 0.00, A 0, B 0, C 0} C_DIS
LIN {X 54.66, Y 162.38, Z 0.00, A 0, B 0, C 0} C_DIS
LIN {X 54.48, Y 162.56, Z 0.00, A 0, B 0, C 0} C_DIS
LIN {X 54.30, Y 162.74, Z 0.00, A 0, B 0, C 0} C_DIS
LIN {X 54.12, Y 162.92, Z 0.00, A 0, B 0, C 0} C_DIS
LIN {X 53.93, Y 163.11, Z 0.00, A 0, B 0, C 0} C_DIS
LIN {X 53.75, Y 163.29, Z 0.00, A 0, B 0, C 0} C_DIS
LIN {X 53.57, Y 163.47, Z 0.00, A 0, B 0, C 0} C_DIS
LIN {X 53.39, Y 163.66, Z 0.00, A 0, B 0, C 0} C_DIS
LIN {X 53.21, Y 163.84, Z 0.00, A 0, B 0, C 0} C_DIS
LIN {X 53.03, Y 164.02, Z 0.00, A 0, B 0, C 0} C_DIS
LIN {X 52.84, Y 164.18, Z 0.00, A 0, B 0, C 0} C_DIS
LIN {X 52.65, Y 164.32, Z 0.00, A 0, B 0, C 0} C_DIS
LIN {X 52.45, Y 164.45, Z 0.00, A 0, B 0, C 0} C_DIS
LIN {X 52.25, Y 164.59, Z 0.00, A 0, B 0, C 0} C_DIS
LIN {X 52.07, Y 164.76, Z 0.00, A 0, B 0, C 0} C_DIS
LIN {X 51.88, Y 164.94, Z 0.00, A 0, B 0, C 0} C_DIS
LIN {X 51.70, Y 165.12, Z 0.00, A 0, B 0, C 0} C_DIS
LIN {X 51.53, Y 165.31, Z 0.00, A 0, B 0, C 0} C_DIS
LIN {X 51.35, Y 165.50, Z 0.00, A 0, B 0, C 0} C_DIS
LIN {X 51.17, Y 165.68, Z 0.00, A 0, B 0, C 0} C_DIS
LIN {X 50.98, Y 165.86, Z 0.00, A 0, B 0, C 0} C_DIS
LIN {X 50.80, Y 166.03, Z 0.00, A 0, B 0, C 0} C_DIS
LIN {X 50.62, Y 166.22, Z 0.00, A 0, B 0, C 0} C_DIS
LIN {X 50.44, Y 166.40, Z 0.00, A 0, B 0, C 0} C_DIS
LIN {X 50.26, Y 166.58, Z 0.00, A 0, B 0, C 0} C_DIS
LIN {X 50.08, Y 166.77, Z 0.00, A 0, B 0, C 0} C_DIS
LIN {X 49.90, Y 166.95, Z 0.00, A 0, B 0, C 0} C_DIS
LIN {X 49.72, Y 167.13, Z 0.00, A 0, B 0, C 0} C_DIS
LIN {X 49.54, Y 167.31, Z 0.00, A 0, B 0, C 0} C_DIS
LIN {X 49.35, Y 167.49, Z 0.00, A 0, B 0, C 0} C_DIS
LIN {X 49.17, Y 167.67, Z 0.00, A 0, B 0, C 0} C_DIS
LIN {X 48.99, Y 167.85, Z 0.00, A 0, B 0, C 0} C_DIS
LIN {X 48.82, Y 168.05, Z 0.00, A 0, B 0, C 0} C_DIS
LIN {X 48.67, Y 168.28, Z 0.00, A 0, B 0, C 0} C_DIS
LIN {X 48.51, Y 168.52, Z 0.00, A 0, B 0, C 0} C_DIS
LIN {X 48.35, Y 168.73, Z 0.00, A 0, B 0, C 0} C_DIS
LIN {X 48.17, Y 168.91, Z 0.00, A 0, B 0, C 0} C_DIS
LIN {X 47.98, Y 169.09, Z 0.00, A 0, B 0, C 0} C_DIS
LIN {X 47.80, Y 169.27, Z 0.00, A 0, B 0, C 0} C_DIS
LIN {X 47.62, Y 169.45, Z 0.00, A 0, B 0, C 0} C_DIS
LIN {X 47.44, Y 169.63, Z 0.00, A 0, B 0, C 0} C_DIS
LIN {X 47.26, Y 169.81, Z 0.00, A 0, B 0, C 0} C_DIS
LIN {X 47.08, Y 170.00, Z 0.00, A 0, B 0, C 0} C_DIS
LIN {X 46.90, Y 170.18, Z 0.00, A 0, B 0, C 0} C_DIS
LIN {X 46.72, Y 170.36, Z 0.00, A 0, B 0, C 0} C_DIS
LIN {X 46.54, Y 170.54, Z 0.00, A 0, B 0, C 0} C_DIS
LIN {X 46.35, Y 170.72, Z 0.00, A 0, B 0, C 0} C_DIS
LIN {X 46.17, Y 170.90, Z 0.00, A 0, B 0, C 0} C_DIS
LIN {X 45.99, Y 171.08, Z 0.00, A 0, B 0, C 0} C_DIS
LIN {X 45.82, Y 171.28, Z 0.00, A 0, B 0, C 0} C_DIS
LIN {X 45.66, Y 171.50, Z 0.00, A 0, B 0, C 0} C_DIS
LIN {X 45.50, Y 171.73, Z 0.00, A 0, B 0, C 0} C_DIS
LIN {X 45.35, Y 171.97, Z 0.00, A 0, B 0, C 0} C_DIS
LIN {X 45.20, Y 172.20, Z 0.00, A 0, B 0, C 0} C_DIS
LIN {X 45.05, Y 172.43, Z 0.00, A 0, B 0, C 0} C_DIS
LIN {X 44.88, Y 172.64, Z 0.00, A 0, B 0, C 0} C_DIS
LIN {X 44.70, Y 172.83, Z 0.00, A 0, B 0, C 0} C_DIS
LIN {X 44.52, Y 173.01, Z 0.00, A 0, B 0, C 0} C_DIS
LIN {X 44.34, Y 173.19, Z 0.00, A 0, B 0, C 0} C_DIS
LIN {X 44.15, Y 173.36, Z 0.00, A 0, B 0, C 0} C_DIS
LIN {X 43.97, Y 173.54, Z 0.00, A 0, B 0, C 0} C_DIS
LIN {X 43.79, Y 173.73, Z 0.00, A 0, B 0, C 0} C_DIS
LIN {X 43.63, Y 173.94, Z 0.00, A 0, B 0, C 0} C_DIS
LIN {X 43.47, Y 174.16, Z 0.00, A 0, B 0, C 0} C_DIS
LIN {X 43.31, Y 174.38, Z 0.00, A 0, B 0, C 0} C_DIS
LIN {X 43.15, Y 174.61, Z 0.00, A 0, B 0, C 0} C_DIS
LIN {X 43.00, Y 174.85, Z 0.00, A 0, B 0, C 0} C_DIS
LIN {X 42.85, Y 175.08, Z 0.00, A 0, B 0, C 0} C_DIS
LIN {X 42.70, Y 175.31, Z 0.00, A 0, B 0, C 0} C_DIS
LIN {X 42.55, Y 175.55, Z 0.00, A 0, B 0, C 0} C_DIS
LIN {X 42.39, Y 175.78, Z 0.00, A 0, B 0, C 0} C_DIS
LIN {X 42.24, Y 176.01, Z 0.00, A 0, B 0, C 0} C_DIS
LIN {X 42.08, Y 176.24, Z 0.00, A 0, B 0, C 0} C_DIS
LIN {X 41.93, Y 176.47, Z 0.00, A 0, B 0, C 0} C_DIS
LIN {X 41.77, Y 176.70, Z 0.00, A 0, B 0, C 0} C_DIS
LIN {X 41.62, Y 176.93, Z 0.00, A 0, B 0, C 0} C_DIS
LIN {X 41.47, Y 177.17, Z 0.00, A 0, B 0, C 0} C_DIS
LIN {X 41.32, Y 177.41, Z 0.00, A 0, B 0, C 0} C_DIS
LIN {X 41.18, Y 177.66, Z 0.00, A 0, B 0, C 0} C_DIS
LIN {X 41.05, Y 177.92, Z 0.00, A 0, B 0, C 0} C_DIS
LIN {X 40.93, Y 178.19, Z 0.00, A 0, B 0, C 0} C_DIS
LIN {X 40.81, Y 178.47, Z 0.00, A 0, B 0, C 0} C_DIS
LIN {X 40.70, Y 178.75, Z 0.00, A 0, B 0, C 0} C_DIS
LIN {X 40.58, Y 179.03, Z 0.00, A 0, B 0, C 0} C_DIS
LIN {X 40.46, Y 179.29, Z 0.00, A 0, B 0, C 0} C_DIS
LIN {X 40.32, Y 179.54, Z 0.00, A 0, B 0, C 0} C_DIS
LIN {X 40.17, Y 179.78, Z 0.00, A 0, B 0, C 0} C_DIS
LIN {X 40.02, Y 180.02, Z 0.00, A 0, B 0, C 0} C_DIS
LIN {X 39.88, Y 180.27, Z 0.00, A 0, B 0, C 0} C_DIS
LIN {X 39.75, Y 180.53, Z 0.00, A 0, B 0, C 0} C_DIS
LIN {X 39.63, Y 180.80, Z 0.00, A 0, B 0, C 0} C_DIS
LIN {X 39.52, Y 181.08, Z 0.00, A 0, B 0, C 0} C_DIS
LIN {X 39.40, Y 181.36, Z 0.00, A 0, B 0, C 0} C_DIS
LIN {X 39.28, Y 181.64, Z 0.00, A 0, B 0, C 0} C_DIS
LIN {X 39.16, Y 181.90, Z 0.00, A 0, B 0, C 0} C_DIS
LIN {X 39.02, Y 182.16, Z 0.00, A 0, B 0, C 0} C_DIS
LIN {X 38.87, Y 182.39, Z 0.00, A 0, B 0, C 0} C_DIS
LIN {X 38.72, Y 182.63, Z 0.00, A 0, B 0, C 0} C_DIS
LIN {X 38.58, Y 182.88, Z 0.00, A 0, B 0, C 0} C_DIS
LIN {X 38.45, Y 183.14, Z 0.00, A 0, B 0, C 0} C_DIS
LIN {X 38.33, Y 183.41, Z 0.00, A 0, B 0, C 0} C_DIS
LIN {X 38.22, Y 183.70, Z 0.00, A 0, B 0, C 0} C_DIS
LIN {X 38.12, Y 183.99, Z 0.00, A 0, B 0, C 0} C_DIS
LIN {X 38.02, Y 184.28, Z 0.00, A 0, B 0, C 0} C_DIS
LIN {X 37.92, Y 184.57, Z 0.00, A 0, B 0, C 0} C_DIS
LIN {X 37.82, Y 184.86, Z 0.00, A 0, B 0, C 0} C_DIS
LIN {X 37.72, Y 185.15, Z 0.00, A 0, B 0, C 0} C_DIS
LIN {X 37.61, Y 185.42, Z 0.00, A 0, B 0, C 0} C_DIS
LIN {X 37.49, Y 185.70, Z 0.00, A 0, B 0, C 0} C_DIS
LIN {X 37.36, Y 185.97, Z 0.00, A 0, B 0, C 0} C_DIS
LIN {X 37.24, Y 186.24, Z 0.00, A 0, B 0, C 0} C_DIS
LIN {X 37.11, Y 186.50, Z 0.00, A 0, B 0, C 0} C_DIS
LIN {X 36.99, Y 186.78, Z 0.00, A 0, B 0, C 0} C_DIS
LIN {X 36.88, Y 187.05, Z 0.00, A 0, B 0, C 0} C_DIS
LIN {X 36.77, Y 187.34, Z 0.00, A 0, B 0, C 0} C_DIS
LIN {X 36.68, Y 187.64, Z 0.00, A 0, B 0, C 0} C_DIS
LIN {X 36.60, Y 187.94, Z 0.00, A 0, B 0, C 0} C_DIS
LIN {X 36.50, Y 188.23, Z 0.00, A 0, B 0, C 0} C_DIS
LIN {X 36.38, Y 188.51, Z 0.00, A 0, B 0, C 0} C_DIS
LIN {X 36.29, Y 188.80, Z 0.00, A 0, B 0, C 0} C_DIS
LIN {X 36.21, Y 189.11, Z 0.00, A 0, B 0, C 0} C_DIS
LIN {X 36.12, Y 189.41, Z 0.00, A 0, B 0, C 0} C_DIS
LIN {X 36.00, Y 189.68, Z 0.00, A 0, B 0, C 0} C_DIS
LIN {X 35.89, Y 189.96, Z 0.00, A 0, B 0, C 0} C_DIS
LIN {X 35.82, Y 190.27, Z 0.00, A 0, B 0, C 0} C_DIS
LIN {X 35.76, Y 190.59, Z 0.00, A 0, B 0, C 0} C_DIS
LIN {X 35.69, Y 190.90, Z 0.00, A 0, B 0, C 0} C_DIS
LIN {X 35.61, Y 191.20, Z 0.00, A 0, B 0, C 0} C_DIS
LIN {X 35.52, Y 191.50, Z 0.00, A 0, B 0, C 0} C_DIS
LIN {X 35.45, Y 191.81, Z 0.00, A 0, B 0, C 0} C_DIS
LIN {X 35.40, Y 192.13, Z 0.00, A 0, B 0, C 0} C_DIS
LIN {X 35.33, Y 192.44, Z 0.00, A 0, B 0, C 0} C_DIS
LIN {X 35.22, Y 192.72, Z 0.00, A 0, B 0, C 0} C_DIS
LIN {X 35.11, Y 193.00, Z 0.00, A 0, B 0, C 0} C_DIS
LIN {X 35.01, Y 193.29, Z 0.00, A 0, B 0, C 0} C_DIS
LIN {X 34.94, Y 193.60, Z 0.00, A 0, B 0, C 0} C_DIS
LIN {X 34.88, Y 193.91, Z 0.00, A 0, B 0, C 0} C_DIS
LIN {X 34.82, Y 194.23, Z 0.00, A 0, B 0, C 0} C_DIS
LIN {X 34.77, Y 194.55, Z 0.00, A 0, B 0, C 0} C_DIS
LIN {X 34.71, Y 194.87, Z 0.00, A 0, B 0, C 0} C_DIS
LIN {X 34.66, Y 195.18, Z 0.00, A 0, B 0, C 0} C_DIS
LIN {X 34.61, Y 195.50, Z 0.00, A 0, B 0, C 0} C_DIS
LIN {X 34.57, Y 195.82, Z 0.00, A 0, B 0, C 0} C_DIS
LIN {X 34.51, Y 196.14, Z 0.00, A 0, B 0, C 0} C_DIS
LIN {X 34.46, Y 196.46, Z 0.00, A 0, B 0, C 0} C_DIS
LIN {X 34.39, Y 196.77, Z 0.00, A 0, B 0, C 0} C_DIS
LIN {X 34.31, Y 197.07, Z 0.00, A 0, B 0, C 0} C_DIS
LIN {X 34.23, Y 197.38, Z 0.00, A 0, B 0, C 0} C_DIS
LIN {X 34.15, Y 197.68, Z 0.00, A 0, B 0, C 0} C_DIS
LIN {X 34.09, Y 197.99, Z 0.00, A 0, B 0, C 0} C_DIS
LIN {X 34.03, Y 198.31, Z 0.00, A 0, B 0, C 0} C_DIS
LIN {X 33.98, Y 198.63, Z 0.00, A 0, B 0, C 0} C_DIS
LIN {X 33.93, Y 198.95, Z 0.00, A 0, B 0, C 0} C_DIS
LIN {X 33.89, Y 199.27, Z 0.00, A 0, B 0, C 0} C_DIS
LIN {X 33.86, Y 199.60, Z 0.00, A 0, B 0, C 0} C_DIS
LIN {X 33.83, Y 199.92, Z 0.00, A 0, B 0, C 0} C_DIS
LIN {X 33.80, Y 200.24, Z 0.00, A 0, B 0, C 0} C_DIS
LIN {X 33.77, Y 200.57, Z 0.00, A 0, B 0, C 0} C_DIS
LIN {X 33.73, Y 200.89, Z 0.00, A 0, B 0, C 0} C_DIS
LIN {X 33.67, Y 201.20, Z 0.00, A 0, B 0, C 0} C_DIS
LIN {X 33.61, Y 201.52, Z 0.00, A 0, B 0, C 0} C_DIS
LIN {X 33.55, Y 201.84, Z 0.00, A 0, B 0, C 0} C_DIS
LIN {X 33.50, Y 202.16, Z 0.00, A 0, B 0, C 0} C_DIS
LIN {X 33.46, Y 202.48, Z 0.00, A 0, B 0, C 0} C_DIS
LIN {X 33.43, Y 202.80, Z 0.00, A 0, B 0, C 0} C_DIS
LIN {X 33.41, Y 203.13, Z 0.00, A 0, B 0, C 0} C_DIS
LIN {X 33.40, Y 203.45, Z 0.00, A 0, B 0, C 0} C_DIS
LIN {X 33.39, Y 203.78, Z 0.00, A 0, B 0, C 0} C_DIS
LIN {X 33.37, Y 204.11, Z 0.00, A 0, B 0, C 0} C_DIS
LIN {X 33.34, Y 204.43, Z 0.00, A 0, B 0, C 0} C_DIS
LIN {X 33.30, Y 204.75, Z 0.00, A 0, B 0, C 0} C_DIS
LIN {X 33.25, Y 205.07, Z 0.00, A 0, B 0, C 0} C_DIS
LIN {X 33.20, Y 205.39, Z 0.00, A 0, B 0, C 0} C_DIS
LIN {X 33.14, Y 205.70, Z 0.00, A 0, B 0, C 0} C_DIS
LIN {X 33.08, Y 206.02, Z 0.00, A 0, B 0, C 0} C_DIS
LIN {X 33.03, Y 206.34, Z 0.00, A 0, B 0, C 0} C_DIS
LIN {X 32.99, Y 206.66, Z 0.00, A 0, B 0, C 0} C_DIS
LIN {X 32.97, Y 206.98, Z 0.00, A 0, B 0, C 0} C_DIS
LIN {X 32.95, Y 207.31, Z 0.00, A 0, B 0, C 0} C_DIS
LIN {X 32.96, Y 207.64, Z 0.00, A 0, B 0, C 0} C_DIS
LIN {X 32.96, Y 207.97, Z 0.00, A 0, B 0, C 0} C_DIS
LIN {X 32.97, Y 208.30, Z 0.00, A 0, B 0, C 0} C_DIS
LIN {X 32.98, Y 208.63, Z 0.00, A 0, B 0, C 0} C_DIS
LIN {X 32.97, Y 208.95, Z 0.00, A 0, B 0, C 0} C_DIS
LIN {X 32.97, Y 209.28, Z 0.00, A 0, B 0, C 0} C_DIS
LIN {X 32.97, Y 209.61, Z 0.00, A 0, B 0, C 0} C_DIS
LIN {X 32.96, Y 209.93, Z 0.00, A 0, B 0, C 0} C_DIS
LIN {X 32.96, Y 210.26, Z 0.00, A 0, B 0, C 0} C_DIS
LIN {X 32.96, Y 210.59, Z 0.00, A 0, B 0, C 0} C_DIS
LIN {X 32.97, Y 210.92, Z 0.00, A 0, B 0, C 0} C_DIS
LIN {X 32.99, Y 211.24, Z 0.00, A 0, B 0, C 0} C_DIS
LIN {X 33.02, Y 211.57, Z 0.00, A 0, B 0, C 0} C_DIS
LIN {X 33.07, Y 211.89, Z 0.00, A 0, B 0, C 0} C_DIS
LIN {X 33.12, Y 212.21, Z 0.00, A 0, B 0, C 0} C_DIS
LIN {X 33.18, Y 212.52, Z 0.00, A 0, B 0, C 0} C_DIS
LIN {X 33.24, Y 212.84, Z 0.00, A 0, B 0, C 0} C_DIS
LIN {X 33.29, Y 213.16, Z 0.00, A 0, B 0, C 0} C_DIS
LIN {X 33.34, Y 213.48, Z 0.00, A 0, B 0, C 0} C_DIS
LIN {X 33.38, Y 213.80, Z 0.00, A 0, B 0, C 0} C_DIS
LIN {X 33.40, Y 214.12, Z 0.00, A 0, B 0, C 0} C_DIS
LIN {X 33.40, Y 214.45, Z 0.00, A 0, B 0, C 0} C_DIS
LIN {X 33.41, Y 214.78, Z 0.00, A 0, B 0, C 0} C_DIS
LIN {X 33.40, Y 215.11, Z 0.00, A 0, B 0, C 0} C_DIS
LIN {X 33.40, Y 215.44, Z 0.00, A 0, B 0, C 0} C_DIS
LIN {X 33.40, Y 215.76, Z 0.00, A 0, B 0, C 0} C_DIS
LIN {X 33.40, Y 216.09, Z 0.00, A 0, B 0, C 0} C_DIS
LIN {X 33.42, Y 216.42, Z 0.00, A 0, B 0, C 0} C_DIS
LIN {X 33.45, Y 216.74, Z 0.00, A 0, B 0, C 0} C_DIS
LIN {X 33.49, Y 217.06, Z 0.00, A 0, B 0, C 0} C_DIS
LIN {X 33.55, Y 217.38, Z 0.00, A 0, B 0, C 0} C_DIS
LIN {X 33.60, Y 217.70, Z 0.00, A 0, B 0, C 0} C_DIS
LIN {X 33.66, Y 218.01, Z 0.00, A 0, B 0, C 0} C_DIS
LIN {X 33.71, Y 218.33, Z 0.00, A 0, B 0, C 0} C_DIS
LIN {X 33.76, Y 218.65, Z 0.00, A 0, B 0, C 0} C_DIS
LIN {X 33.80, Y 218.97, Z 0.00, A 0, B 0, C 0} C_DIS
LIN {X 33.83, Y 219.29, Z 0.00, A 0, B 0, C 0} C_DIS
LIN {X 33.86, Y 219.62, Z 0.00, A 0, B 0, C 0} C_DIS
LIN {X 33.89, Y 219.94, Z 0.00, A 0, B 0, C 0} C_DIS
LIN {X 33.92, Y 220.27, Z 0.00, A 0, B 0, C 0} C_DIS
LIN {X 33.96, Y 220.59, Z 0.00, A 0, B 0, C 0} C_DIS
LIN {X 34.01, Y 220.91, Z 0.00, A 0, B 0, C 0} C_DIS
LIN {X 34.07, Y 221.22, Z 0.00, A 0, B 0, C 0} C_DIS
LIN {X 34.14, Y 221.54, Z 0.00, A 0, B 0, C 0} C_DIS
LIN {X 34.21, Y 221.84, Z 0.00, A 0, B 0, C 0} C_DIS
LIN {X 34.29, Y 222.15, Z 0.00, A 0, B 0, C 0} C_DIS
LIN {X 34.38, Y 222.45, Z 0.00, A 0, B 0, C 0} C_DIS
LIN {X 34.45, Y 222.76, Z 0.00, A 0, B 0, C 0} C_DIS
LIN {X 34.50, Y 223.08, Z 0.00, A 0, B 0, C 0} C_DIS
LIN {X 34.54, Y 223.40, Z 0.00, A 0, B 0, C 0} C_DIS
LIN {X 34.61, Y 223.71, Z 0.00, A 0, B 0, C 0} C_DIS
LIN {X 34.70, Y 224.01, Z 0.00, A 0, B 0, C 0} C_DIS
LIN {X 34.79, Y 224.31, Z 0.00, A 0, B 0, C 0} C_DIS
LIN {X 34.86, Y 224.62, Z 0.00, A 0, B 0, C 0} C_DIS
LIN {X 34.92, Y 224.93, Z 0.00, A 0, B 0, C 0} C_DIS
LIN {X 34.97, Y 225.25, Z 0.00, A 0, B 0, C 0} C_DIS
LIN {X 35.02, Y 225.57, Z 0.00, A 0, B 0, C 0} C_DIS
LIN {X 35.10, Y 225.87, Z 0.00, A 0, B 0, C 0} C_DIS
LIN {X 35.19, Y 226.17, Z 0.00, A 0, B 0, C 0} C_DIS
LIN {X 35.27, Y 226.47, Z 0.00, A 0, B 0, C 0} C_DIS
LIN {X 35.33, Y 226.79, Z 0.00, A 0, B 0, C 0} C_DIS
LIN {X 35.39, Y 227.11, Z 0.00, A 0, B 0, C 0} C_DIS
LIN {X 35.47, Y 227.41, Z 0.00, A 0, B 0, C 0} C_DIS
LIN {X 35.59, Y 227.68, Z 0.00, A 0, B 0, C 0} C_DIS
LIN {X 35.70, Y 227.96, Z 0.00, A 0, B 0, C 0} C_DIS
LIN {X 35.78, Y 228.27, Z 0.00, A 0, B 0, C 0} C_DIS
LIN {X 35.87, Y 228.57, Z 0.00, A 0, B 0, C 0} C_DIS
LIN {X 35.98, Y 228.85, Z 0.00, A 0, B 0, C 0} C_DIS
LIN {X 36.08, Y 229.14, Z 0.00, A 0, B 0, C 0} C_DIS
LIN {X 36.17, Y 229.44, Z 0.00, A 0, B 0, C 0} C_DIS
LIN {X 36.26, Y 229.74, Z 0.00, A 0, B 0, C 0} C_DIS
LIN {X 36.36, Y 230.02, Z 0.00, A 0, B 0, C 0} C_DIS
LIN {X 36.47, Y 230.31, Z 0.00, A 0, B 0, C 0} C_DIS
LIN {X 36.57, Y 230.60, Z 0.00, A 0, B 0, C 0} C_DIS
LIN {X 36.65, Y 230.90, Z 0.00, A 0, B 0, C 0} C_DIS
LIN {X 36.74, Y 231.20, Z 0.00, A 0, B 0, C 0} C_DIS
LIN {X 36.84, Y 231.49, Z 0.00, A 0, B 0, C 0} C_DIS
LIN {X 36.96, Y 231.76, Z 0.00, A 0, B 0, C 0} C_DIS
LIN {X 37.05, Y 232.06, Z 0.00, A 0, B 0, C 0} C_DIS
LIN {X 37.13, Y 232.36, Z 0.00, A 0, B 0, C 0} C_DIS
LIN {X 37.22, Y 232.66, Z 0.00, A 0, B 0, C 0} C_DIS
LIN {X 37.34, Y 232.94, Z 0.00, A 0, B 0, C 0} C_DIS
LIN {X 37.45, Y 233.22, Z 0.00, A 0, B 0, C 0} C_DIS
LIN {X 37.52, Y 233.53, Z 0.00, A 0, B 0, C 0} C_DIS
LIN {X 37.61, Y 233.83, Z 0.00, A 0, B 0, C 0} C_DIS
LIN {X 37.72, Y 234.11, Z 0.00, A 0, B 0, C 0} C_DIS
LIN {X 37.83, Y 234.39, Z 0.00, A 0, B 0, C 0} C_DIS
LIN {X 37.95, Y 234.66, Z 0.00, A 0, B 0, C 0} C_DIS
LIN {X 38.07, Y 234.94, Z 0.00, A 0, B 0, C 0} C_DIS
LIN {X 38.19, Y 235.21, Z 0.00, A 0, B 0, C 0} C_DIS
LIN {X 38.31, Y 235.48, Z 0.00, A 0, B 0, C 0} C_DIS
LIN {X 38.43, Y 235.76, Z 0.00, A 0, B 0, C 0} C_DIS
LIN {X 38.55, Y 236.03, Z 0.00, A 0, B 0, C 0} C_DIS
LIN {X 38.68, Y 236.30, Z 0.00, A 0, B 0, C 0} C_DIS
LIN {X 38.80, Y 236.57, Z 0.00, A 0, B 0, C 0} C_DIS
LIN {X 38.92, Y 236.84, Z 0.00, A 0, B 0, C 0} C_DIS
LIN {X 39.04, Y 237.11, Z 0.00, A 0, B 0, C 0} C_DIS
LIN {X 39.16, Y 237.38, Z 0.00, A 0, B 0, C 0} C_DIS
LIN {X 39.28, Y 237.66, Z 0.00, A 0, B 0, C 0} C_DIS
LIN {X 39.40, Y 237.94, Z 0.00, A 0, B 0, C 0} C_DIS
LIN {X 39.51, Y 238.21, Z 0.00, A 0, B 0, C 0} C_DIS
LIN {X 39.63, Y 238.49, Z 0.00, A 0, B 0, C 0} C_DIS
LIN {X 39.76, Y 238.76, Z 0.00, A 0, B 0, C 0} C_DIS
LIN {X 39.89, Y 239.02, Z 0.00, A 0, B 0, C 0} C_DIS
LIN {X 40.03, Y 239.27, Z 0.00, A 0, B 0, C 0} C_DIS
LIN {X 40.17, Y 239.51, Z 0.00, A 0, B 0, C 0} C_DIS
LIN {X 40.32, Y 239.75, Z 0.00, A 0, B 0, C 0} C_DIS
LIN {X 40.48, Y 239.98, Z 0.00, A 0, B 0, C 0} C_DIS
LIN {X 40.64, Y 240.20, Z 0.00, A 0, B 0, C 0} C_DIS
LIN {X 40.79, Y 240.43, Z 0.00, A 0, B 0, C 0} C_DIS
LIN {X 40.95, Y 240.66, Z 0.00, A 0, B 0, C 0} C_DIS
LIN {X 41.10, Y 240.90, Z 0.00, A 0, B 0, C 0} C_DIS
LIN {X 41.24, Y 241.15, Z 0.00, A 0, B 0, C 0} C_DIS
LIN {X 41.37, Y 241.40, Z 0.00, A 0, B 0, C 0} C_DIS
LIN {X 41.50, Y 241.67, Z 0.00, A 0, B 0, C 0} C_DIS
LIN {X 41.62, Y 241.94, Z 0.00, A 0, B 0, C 0} C_DIS
LIN {X 41.73, Y 242.22, Z 0.00, A 0, B 0, C 0} C_DIS
LIN {X 41.85, Y 242.50, Z 0.00, A 0, B 0, C 0} C_DIS
LIN {X 41.97, Y 242.78, Z 0.00, A 0, B 0, C 0} C_DIS
LIN {X 42.10, Y 243.04, Z 0.00, A 0, B 0, C 0} C_DIS
LIN {X 42.24, Y 243.28, Z 0.00, A 0, B 0, C 0} C_DIS
LIN {X 42.39, Y 243.51, Z 0.00, A 0, B 0, C 0} C_DIS
LIN {X 42.55, Y 243.74, Z 0.00, A 0, B 0, C 0} C_DIS
LIN {X 42.70, Y 243.98, Z 0.00, A 0, B 0, C 0} C_DIS
LIN {X 42.85, Y 244.22, Z 0.00, A 0, B 0, C 0} C_DIS
LIN {X 43.01, Y 244.45, Z 0.00, A 0, B 0, C 0} C_DIS
LIN {X 43.17, Y 244.66, Z 0.00, A 0, B 0, C 0} C_DIS
LIN {X 43.34, Y 244.87, Z 0.00, A 0, B 0, C 0} C_DIS
LIN {X 43.51, Y 245.06, Z 0.00, A 0, B 0, C 0} C_DIS
LIN {X 43.69, Y 245.24, Z 0.00, A 0, B 0, C 0} C_DIS
LIN {X 43.88, Y 245.42, Z 0.00, A 0, B 0, C 0} C_DIS
LIN {X 44.06, Y 245.59, Z 0.00, A 0, B 0, C 0} C_DIS
LIN {X 44.24, Y 245.77, Z 0.00, A 0, B 0, C 0} C_DIS
LIN {X 44.42, Y 245.96, Z 0.00, A 0, B 0, C 0} C_DIS
LIN {X 44.59, Y 246.17, Z 0.00, A 0, B 0, C 0} C_DIS
LIN {X 44.75, Y 246.39, Z 0.00, A 0, B 0, C 0} C_DIS
LIN {X 44.90, Y 246.62, Z 0.00, A 0, B 0, C 0} C_DIS
LIN {X 45.05, Y 246.87, Z 0.00, A 0, B 0, C 0} C_DIS
LIN {X 45.20, Y 247.10, Z 0.00, A 0, B 0, C 0} C_DIS
LIN {X 45.36, Y 247.32, Z 0.00, A 0, B 0, C 0} C_DIS
LIN {X 45.53, Y 247.52, Z 0.00, A 0, B 0, C 0} C_DIS
LIN {X 45.71, Y 247.71, Z 0.00, A 0, B 0, C 0} C_DIS
LIN {X 45.89, Y 247.88, Z 0.00, A 0, B 0, C 0} C_DIS
LIN {X 46.08, Y 248.06, Z 0.00, A 0, B 0, C 0} C_DIS
LIN {X 46.26, Y 248.23, Z 0.00, A 0, B 0, C 0} C_DIS
LIN {X 46.44, Y 248.41, Z 0.00, A 0, B 0, C 0} C_DIS
LIN {X 46.62, Y 248.61, Z 0.00, A 0, B 0, C 0} C_DIS
LIN {X 46.78, Y 248.82, Z 0.00, A 0, B 0, C 0} C_DIS
LIN {X 46.94, Y 249.05, Z 0.00, A 0, B 0, C 0} C_DIS
LIN {X 47.10, Y 249.27, Z 0.00, A 0, B 0, C 0} C_DIS
LIN {X 47.26, Y 249.48, Z 0.00, A 0, B 0, C 0} C_DIS
LIN {X 47.44, Y 249.67, Z 0.00, A 0, B 0, C 0} C_DIS
LIN {X 47.63, Y 249.84, Z 0.00, A 0, B 0, C 0} C_DIS
LIN {X 47.81, Y 250.01, Z 0.00, A 0, B 0, C 0} C_DIS
LIN {X 48.00, Y 250.17, Z 0.00, A 0, B 0, C 0} C_DIS
LIN {X 48.19, Y 250.32, Z 0.00, A 0, B 0, C 0} C_DIS
LIN {X 48.39, Y 250.45, Z 0.00, A 0, B 0, C 0} C_DIS
LIN {X 48.59, Y 250.59, Z 0.00, A 0, B 0, C 0} C_DIS
LIN {X 48.78, Y 250.75, Z 0.00, A 0, B 0, C 0} C_DIS
LIN {X 48.96, Y 250.94, Z 0.00, A 0, B 0, C 0} C_DIS
LIN {X 49.14, Y 251.12, Z 0.00, A 0, B 0, C 0} C_DIS
LIN {X 49.31, Y 251.32, Z 0.00, A 0, B 0, C 0} C_DIS
LIN {X 49.49, Y 251.51, Z 0.00, A 0, B 0, C 0} C_DIS
LIN {X 49.67, Y 251.69, Z 0.00, A 0, B 0, C 0} C_DIS
LIN {X 49.85, Y 251.87, Z 0.00, A 0, B 0, C 0} C_DIS
LIN {X 50.04, Y 252.03, Z 0.00, A 0, B 0, C 0} C_DIS
LIN {X 50.24, Y 252.17, Z 0.00, A 0, B 0, C 0} C_DIS
LIN {X 50.43, Y 252.31, Z 0.00, A 0, B 0, C 0} C_DIS
LIN {X 50.63, Y 252.45, Z 0.00, A 0, B 0, C 0} C_DIS
LIN {X 50.82, Y 252.61, Z 0.00, A 0, B 0, C 0} C_DIS
LIN {X 51.01, Y 252.77, Z 0.00, A 0, B 0, C 0} C_DIS
LIN {X 51.20, Y 252.91, Z 0.00, A 0, B 0, C 0} C_DIS
LIN {X 51.40, Y 253.04, Z 0.00, A 0, B 0, C 0} C_DIS
LIN {X 51.60, Y 253.18, Z 0.00, A 0, B 0, C 0} C_DIS
LIN {X 51.79, Y 253.34, Z 0.00, A 0, B 0, C 0} C_DIS
LIN {X 51.98, Y 253.50, Z 0.00, A 0, B 0, C 0} C_DIS
LIN {X 52.17, Y 253.64, Z 0.00, A 0, B 0, C 0} C_DIS
LIN {X 52.38, Y 253.75, Z 0.00, A 0, B 0, C 0} C_DIS
LIN {X 52.56, Y 253.92, Z 0.00, A 0, B 0, C 0} C_DIS
LIN {X 52.75, Y 254.10, Z 0.00, A 0, B 0, C 0} C_DIS
LIN {X 52.95, Y 254.22, Z 0.00, A 0, B 0, C 0} C_DIS
LIN {X 53.16, Y 254.32, Z 0.00, A 0, B 0, C 0} C_DIS
LIN {X 53.36, Y 254.41, Z 0.00, A 0, B 0, C 0} C_DIS
LIN {X 53.57, Y 254.52, Z 0.00, A 0, B 0, C 0} C_DIS
LIN {X 53.77, Y 254.66, Z 0.00, A 0, B 0, C 0} C_DIS
LIN {X 53.97, Y 254.79, Z 0.00, A 0, B 0, C 0} C_DIS
LIN {X 54.18, Y 254.87, Z 0.00, A 0, B 0, C 0} C_DIS
LIN {X 54.39, Y 254.94, Z 0.00, A 0, B 0, C 0} C_DIS
LIN {X 54.60, Y 255.03, Z 0.00, A 0, B 0, C 0} C_DIS
LIN {X 54.80, Y 255.13, Z 0.00, A 0, B 0, C 0} C_DIS
LIN {X 55.00, Y 255.26, Z 0.00, A 0, B 0, C 0} C_DIS
LIN {X 55.20, Y 255.40, Z 0.00, A 0, B 0, C 0} C_DIS
LIN {X 55.41, Y 255.50, Z 0.00, A 0, B 0, C 0} C_DIS
LIN {X 55.62, Y 255.57, Z 0.00, A 0, B 0, C 0} C_DIS
LIN {X 55.83, Y 255.65, Z 0.00, A 0, B 0, C 0} C_DIS
LIN {X 56.04, Y 255.75, Z 0.00, A 0, B 0, C 0} C_DIS
LIN {X 56.24, Y 255.87, Z 0.00, A 0, B 0, C 0} C_DIS
LIN {X 56.44, Y 256.01, Z 0.00, A 0, B 0, C 0} C_DIS
LIN {X 56.64, Y 256.13, Z 0.00, A 0, B 0, C 0} C_DIS
LIN {X 56.85, Y 256.21, Z 0.00, A 0, B 0, C 0} C_DIS
LIN {X 57.06, Y 256.29, Z 0.00, A 0, B 0, C 0} C_DIS
LIN {X 57.27, Y 256.37, Z 0.00, A 0, B 0, C 0} C_DIS
LIN {X 57.48, Y 256.44, Z 0.00, A 0, B 0, C 0} C_DIS
LIN {X 57.70, Y 256.51, Z 0.00, A 0, B 0, C 0} C_DIS
LIN {X 57.91, Y 256.59, Z 0.00, A 0, B 0, C 0} C_DIS
LIN {X 58.12, Y 256.67, Z 0.00, A 0, B 0, C 0} C_DIS
LIN {X 58.33, Y 256.76, Z 0.00, A 0, B 0, C 0} C_DIS
LIN {X 58.54, Y 256.84, Z 0.00, A 0, B 0, C 0} C_DIS
LIN {X 58.75, Y 256.93, Z 0.00, A 0, B 0, C 0} C_DIS
LIN {X 58.96, Y 257.02, Z 0.00, A 0, B 0, C 0} C_DIS
LIN {X 59.17, Y 257.09, Z 0.00, A 0, B 0, C 0} C_DIS
LIN {X 59.38, Y 257.15, Z 0.00, A 0, B 0, C 0} C_DIS
LIN {X 59.60, Y 257.18, Z 0.00, A 0, B 0, C 0} C_DIS
LIN {X 59.82, Y 257.21, Z 0.00, A 0, B 0, C 0} C_DIS
LIN {X 60.03, Y 257.23, Z 0.00, A 0, B 0, C 0} C_DIS
LIN {X 60.25, Y 257.25, Z 0.00, A 0, B 0, C 0} C_DIS
LIN {X 60.46, Y 257.27, Z 0.00, A 0, B 0, C 0} C_DIS
LIN {X 60.68, Y 257.32, Z 0.00, A 0, B 0, C 0} C_DIS
LIN {X 60.89, Y 257.38, Z 0.00, A 0, B 0, C 0} C_DIS
LIN {X 61.10, Y 257.46, Z 0.00, A 0, B 0, C 0} C_DIS
LIN {X 61.31, Y 257.56, Z 0.00, A 0, B 0, C 0} C_DIS
LIN {X 61.52, Y 257.65, Z 0.00, A 0, B 0, C 0} C_DIS
LIN {X 61.73, Y 257.74, Z 0.00, A 0, B 0, C 0} C_DIS
LIN {X 61.95, Y 257.80, Z 0.00, A 0, B 0, C 0} C_DIS
LIN {X 62.16, Y 257.84, Z 0.00, A 0, B 0, C 0} C_DIS
LIN {X 62.38, Y 257.86, Z 0.00, A 0, B 0, C 0} C_DIS
LIN {X 62.59, Y 257.88, Z 0.00, A 0, B 0, C 0} C_DIS
LIN {X 62.81, Y 257.89, Z 0.00, A 0, B 0, C 0} C_DIS
LIN {X 63.03, Y 257.89, Z 0.00, A 0, B 0, C 0} C_DIS
LIN {X 63.25, Y 257.89, Z 0.00, A 0, B 0, C 0} C_DIS
LIN {X 63.46, Y 257.88, Z 0.00, A 0, B 0, C 0} C_DIS
LIN {X 63.68, Y 257.88, Z 0.00, A 0, B 0, C 0} C_DIS
LIN {X 63.90, Y 257.88, Z 0.00, A 0, B 0, C 0} C_DIS
LIN {X 64.12, Y 257.88, Z 0.00, A 0, B 0, C 0} C_DIS
LIN {X 64.33, Y 257.88, Z 0.00, A 0, B 0, C 0} C_DIS
LIN {X 64.55, Y 257.88, Z 0.00, A 0, B 0, C 0} C_DIS
LIN {X 64.77, Y 257.88, Z 0.00, A 0, B 0, C 0} C_DIS
LIN {X 64.99, Y 257.88, Z 0.00, A 0, B 0, C 0} C_DIS
LIN {X 65.20, Y 257.88, Z 0.00, A 0, B 0, C 0} C_DIS
LIN {X 65.42, Y 257.88, Z 0.00, A 0, B 0, C 0} C_DIS
LIN {X 65.64, Y 257.88, Z 0.00, A 0, B 0, C 0} C_DIS
LIN {X 65.86, Y 257.88, Z 0.00, A 0, B 0, C 0} C_DIS
LIN {X 66.07, Y 257.88, Z 0.00, A 0, B 0, C 0} C_DIS
LIN {X 66.29, Y 257.88, Z 0.00, A 0, B 0, C 0} C_DIS
LIN {X 66.51, Y 257.88, Z 0.00, A 0, B 0, C 0} C_DIS
LIN {X 66.73, Y 257.88, Z 0.00, A 0, B 0, C 0} C_DIS
LIN {X 66.94, Y 257.88, Z 0.00, A 0, B 0, C 0} C_DIS
LIN {X 67.16, Y 257.88, Z 0.00, A 0, B 0, C 0} C_DIS
LIN {X 67.38, Y 257.88, Z 0.00, A 0, B 0, C 0} C_DIS
LIN {X 67.60, Y 257.88, Z 0.00, A 0, B 0, C 0} C_DIS
LIN {X 67.81, Y 257.88, Z 0.00, A 0, B 0, C 0} C_DIS
LIN {X 68.03, Y 257.88, Z 0.00, A 0, B 0, C 0} C_DIS
LIN {X 68.25, Y 257.88, Z 0.00, A 0, B 0, C 0} C_DIS
LIN {X 68.47, Y 257.88, Z 0.00, A 0, B 0, C 0} C_DIS
LIN {X 68.68, Y 257.88, Z 0.00, A 0, B 0, C 0} C_DIS
LIN {X 68.90, Y 257.88, Z 0.00, A 0, B 0, C 0} C_DIS
LIN {X 69.12, Y 257.88, Z 0.00, A 0, B 0, C 0} C_DIS
LIN {X 69.33, Y 257.88, Z 0.00, A 0, B 0, C 0} C_DIS
LIN {X 69.55, Y 257.88, Z 0.00, A 0, B 0, C 0} C_DIS
LIN {X 69.77, Y 257.88, Z 0.00, A 0, B 0, C 0} C_DIS
LIN {X 69.99, Y 257.88, Z 0.00, A 0, B 0, C 0} C_DIS
LIN {X 70.20, Y 257.88, Z 0.00, A 0, B 0, C 0} C_DIS
LIN {X 70.42, Y 257.88, Z 0.00, A 0, B 0, C 0} C_DIS
LIN {X 70.64, Y 257.88, Z 0.00, A 0, B 0, C 0} C_DIS
LIN {X 70.86, Y 257.88, Z 0.00, A 0, B 0, C 0} C_DIS
LIN {X 71.07, Y 257.88, Z 0.00, A 0, B 0, C 0} C_DIS
LIN {X 71.29, Y 257.88, Z 0.00, A 0, B 0, C 0} C_DIS
LIN {X 71.51, Y 257.88, Z 0.00, A 0, B 0, C 0} C_DIS
LIN {X 71.73, Y 257.88, Z 0.00, A 0, B 0, C 0} C_DIS
LIN {X 71.94, Y 257.88, Z 0.00, A 0, B 0, C 0} C_DIS
LIN {X 72.16, Y 257.88, Z 0.00, A 0, B 0, C 0} C_DIS
LIN {X 72.38, Y 257.88, Z 0.00, A 0, B 0, C 0} C_DIS
LIN {X 72.60, Y 257.88, Z 0.00, A 0, B 0, C 0} C_DIS
LIN {X 72.81, Y 257.88, Z 0.00, A 0, B 0, C 0} C_DIS
LIN {X 73.03, Y 257.88, Z 0.00, A 0, B 0, C 0} C_DIS
LIN {X 73.25, Y 257.88, Z 0.00, A 0, B 0, C 0} C_DIS
LIN {X 73.47, Y 257.88, Z 0.00, A 0, B 0, C 0} C_DIS
LIN {X 73.68, Y 257.88, Z 0.00, A 0, B 0, C 0} C_DIS
LIN {X 73.90, Y 257.88, Z 0.00, A 0, B 0, C 0} C_DIS
LIN {X 74.12, Y 257.88, Z 0.00, A 0, B 0, C 0} C_DIS
LIN {X 74.34, Y 257.88, Z 0.00, A 0, B 0, C 0} C_DIS
LIN {X 74.55, Y 257.88, Z 0.00, A 0, B 0, C 0} C_DIS
LIN {X 74.77, Y 257.88, Z 0.00, A 0, B 0, C 0} C_DIS
LIN {X 74.99, Y 257.88, Z 0.00, A 0, B 0, C 0} C_DIS
LIN {X 75.21, Y 257.88, Z 0.00, A 0, B 0, C 0} C_DIS
LIN {X 75.42, Y 257.88, Z 0.00, A 0, B 0, C 0} C_DIS
LIN {X 75.64, Y 257.88, Z 0.00, A 0, B 0, C 0} C_DIS
LIN {X 75.86, Y 257.88, Z 0.00, A 0, B 0, C 0} C_DIS
LIN {X 76.08, Y 257.88, Z 0.00, A 0, B 0, C 0} C_DIS
LIN {X 76.29, Y 257.88, Z 0.00, A 0, B 0, C 0} C_DIS
LIN {X 76.51, Y 257.88, Z 0.00, A 0, B 0, C 0} C_DIS
LIN {X 76.73, Y 257.88, Z 0.00, A 0, B 0, C 0} C_DIS
LIN {X 76.95, Y 257.88, Z 0.00, A 0, B 0, C 0} C_DIS
LIN {X 77.16, Y 257.88, Z 0.00, A 0, B 0, C 0} C_DIS
LIN {X 77.38, Y 257.88, Z 0.00, A 0, B 0, C 0} C_DIS
LIN {X 77.60, Y 257.88, Z 0.00, A 0, B 0, C 0} C_DIS
LIN {X 77.82, Y 257.88, Z 0.00, A 0, B 0, C 0} C_DIS
LIN {X 78.03, Y 257.88, Z 0.00, A 0, B 0, C 0} C_DIS
LIN {X 78.25, Y 257.88, Z 0.00, A 0, B 0, C 0} C_DIS
LIN {X 78.47, Y 257.88, Z 0.00, A 0, B 0, C 0} C_DIS
LIN {X 78.69, Y 257.88, Z 0.00, A 0, B 0, C 0} C_DIS
LIN {X 78.90, Y 257.88, Z 0.00, A 0, B 0, C 0} C_DIS
LIN {X 79.12, Y 257.88, Z 0.00, A 0, B 0, C 0} C_DIS
LIN {X 79.34, Y 257.88, Z 0.00, A 0, B 0, C 0} C_DIS
LIN {X 79.56, Y 257.88, Z 0.00, A 0, B 0, C 0} C_DIS
LIN {X 79.77, Y 257.88, Z 0.00, A 0, B 0, C 0} C_DIS
LIN {X 79.99, Y 257.88, Z 0.00, A 0, B 0, C 0} C_DIS
LIN {X 80.21, Y 257.88, Z 0.00, A 0, B 0, C 0} C_DIS
LIN {X 80.43, Y 257.88, Z 0.00, A 0, B 0, C 0} C_DIS
LIN {X 80.64, Y 257.88, Z 0.00, A 0, B 0, C 0} C_DIS
LIN {X 80.86, Y 257.88, Z 0.00, A 0, B 0, C 0} C_DIS
LIN {X 81.08, Y 257.88, Z 0.00, A 0, B 0, C 0} C_DIS
LIN {X 81.30, Y 257.88, Z 0.00, A 0, B 0, C 0} C_DIS
LIN {X 81.51, Y 257.88, Z 0.00, A 0, B 0, C 0} C_DIS
LIN {X 81.73, Y 257.88, Z 0.00, A 0, B 0, C 0} C_DIS
LIN {X 81.95, Y 257.88, Z 0.00, A 0, B 0, C 0} C_DIS
LIN {X 82.16, Y 257.88, Z 0.00, A 0, B 0, C 0} C_DIS
LIN {X 82.38, Y 257.88, Z 0.00, A 0, B 0, C 0} C_DIS
LIN {X 82.60, Y 257.88, Z 0.00, A 0, B 0, C 0} C_DIS
LIN {X 82.82, Y 257.88, Z 0.00, A 0, B 0, C 0} C_DIS
LIN {X 83.03, Y 257.88, Z 0.00, A 0, B 0, C 0} C_DIS
LIN {X 83.25, Y 257.88, Z 0.00, A 0, B 0, C 0} C_DIS
LIN {X 83.47, Y 257.88, Z 0.00, A 0, B 0, C 0} C_DIS
LIN {X 83.69, Y 257.88, Z 0.00, A 0, B 0, C 0} C_DIS
LIN {X 83.90, Y 257.88, Z 0.00, A 0, B 0, C 0} C_DIS
LIN {X 84.12, Y 257.88, Z 0.00, A 0, B 0, C 0} C_DIS
LIN {X 84.34, Y 257.88, Z 0.00, A 0, B 0, C 0} C_DIS
LIN {X 84.56, Y 257.88, Z 0.00, A 0, B 0, C 0} C_DIS
LIN {X 84.77, Y 257.88, Z 0.00, A 0, B 0, C 0} C_DIS
LIN {X 84.99, Y 257.88, Z 0.00, A 0, B 0, C 0} C_DIS
LIN {X 85.21, Y 257.88, Z 0.00, A 0, B 0, C 0} C_DIS
LIN {X 85.43, Y 257.88, Z 0.00, A 0, B 0, C 0} C_DIS
LIN {X 85.64, Y 257.88, Z 0.00, A 0, B 0, C 0} C_DIS
LIN {X 85.86, Y 257.88, Z 0.00, A 0, B 0, C 0} C_DIS
LIN {X 86.08, Y 257.88, Z 0.00, A 0, B 0, C 0} C_DIS
LIN {X 86.30, Y 257.88, Z 0.00, A 0, B 0, C 0} C_DIS
LIN {X 86.51, Y 257.88, Z 0.00, A 0, B 0, C 0} C_DIS
LIN {X 86.73, Y 257.88, Z 0.00, A 0, B 0, C 0} C_DIS
LIN {X 86.95, Y 257.88, Z 0.00, A 0, B 0, C 0} C_DIS
LIN {X 87.17, Y 257.88, Z 0.00, A 0, B 0, C 0} C_DIS
LIN {X 87.38, Y 257.88, Z 0.00, A 0, B 0, C 0} C_DIS
LIN {X 87.60, Y 257.88, Z 0.00, A 0, B 0, C 0} C_DIS
LIN {X 87.82, Y 257.88, Z 0.00, A 0, B 0, C 0} C_DIS
LIN {X 88.04, Y 257.88, Z 0.00, A 0, B 0, C 0} C_DIS
LIN {X 88.25, Y 257.88, Z 0.00, A 0, B 0, C 0} C_DIS
LIN {X 88.47, Y 257.88, Z 0.00, A 0, B 0, C 0} C_DIS
LIN {X 88.69, Y 257.88, Z 0.00, A 0, B 0, C 0} C_DIS
LIN {X 88.91, Y 257.88, Z 0.00, A 0, B 0, C 0} C_DIS
LIN {X 89.12, Y 257.88, Z 0.00, A 0, B 0, C 0} C_DIS
LIN {X 89.34, Y 257.88, Z 0.00, A 0, B 0, C 0} C_DIS
LIN {X 89.56, Y 257.88, Z 0.00, A 0, B 0, C 0} C_DIS
LIN {X 89.78, Y 257.88, Z 0.00, A 0, B 0, C 0} C_DIS
LIN {X 89.99, Y 257.88, Z 0.00, A 0, B 0, C 0} C_DIS
LIN {X 90.21, Y 257.88, Z 0.00, A 0, B 0, C 0} C_DIS
LIN {X 90.43, Y 257.88, Z 0.00, A 0, B 0, C 0} C_DIS
LIN {X 90.65, Y 257.88, Z 0.00, A 0, B 0, C 0} C_DIS
LIN {X 90.86, Y 257.88, Z 0.00, A 0, B 0, C 0} C_DIS
LIN {X 91.08, Y 257.88, Z 0.00, A 0, B 0, C 0} C_DIS
LIN {X 91.30, Y 257.88, Z 0.00, A 0, B 0, C 0} C_DIS
LIN {X 91.52, Y 257.88, Z 0.00, A 0, B 0, C 0} C_DIS
LIN {X 91.73, Y 257.88, Z 0.00, A 0, B 0, C 0} C_DIS
LIN {X 91.95, Y 257.88, Z 0.00, A 0, B 0, C 0} C_DIS
LIN {X 92.17, Y 257.88, Z 0.00, A 0, B 0, C 0} C_DIS
LIN {X 92.39, Y 257.88, Z 0.00, A 0, B 0, C 0} C_DIS
LIN {X 92.60, Y 257.88, Z 0.00, A 0, B 0, C 0} C_DIS
LIN {X 92.82, Y 257.88, Z 0.00, A 0, B 0, C 0} C_DIS
LIN {X 93.04, Y 257.88, Z 0.00, A 0, B 0, C 0} C_DIS
LIN {X 93.26, Y 257.88, Z 0.00, A 0, B 0, C 0} C_DIS
LIN {X 93.47, Y 257.88, Z 0.00, A 0, B 0, C 0} C_DIS
LIN {X 93.69, Y 257.88, Z 0.00, A 0, B 0, C 0} C_DIS
LIN {X 93.91, Y 257.88, Z 0.00, A 0, B 0, C 0} C_DIS
LIN {X 94.12, Y 257.88, Z 0.00, A 0, B 0, C 0} C_DIS
LIN {X 94.34, Y 257.88, Z 0.00, A 0, B 0, C 0} C_DIS
LIN {X 94.56, Y 257.88, Z 0.00, A 0, B 0, C 0} C_DIS
LIN {X 94.78, Y 257.88, Z 0.00, A 0, B 0, C 0} C_DIS
LIN {X 94.99, Y 257.88, Z 0.00, A 0, B 0, C 0} C_DIS
LIN {X 95.21, Y 257.88, Z 0.00, A 0, B 0, C 0} C_DIS
LIN {X 95.43, Y 257.88, Z 0.00, A 0, B 0, C 0} C_DIS
LIN {X 95.65, Y 257.88, Z 0.00, A 0, B 0, C 0} C_DIS
LIN {X 95.86, Y 257.88, Z 0.00, A 0, B 0, C 0} C_DIS
LIN {X 96.08, Y 257.88, Z 0.00, A 0, B 0, C 0} C_DIS
LIN {X 96.30, Y 257.88, Z 0.00, A 0, B 0, C 0} C_DIS
LIN {X 96.52, Y 257.88, Z 0.00, A 0, B 0, C 0} C_DIS
LIN {X 96.73, Y 257.88, Z 0.00, A 0, B 0, C 0} C_DIS
LIN {X 96.95, Y 257.88, Z 0.00, A 0, B 0, C 0} C_DIS
LIN {X 97.17, Y 257.88, Z 0.00, A 0, B 0, C 0} C_DIS
LIN {X 97.39, Y 257.88, Z 0.00, A 0, B 0, C 0} C_DIS
LIN {X 97.60, Y 257.88, Z 0.00, A 0, B 0, C 0} C_DIS
LIN {X 97.82, Y 257.88, Z 0.00, A 0, B 0, C 0} C_DIS
LIN {X 98.04, Y 257.88, Z 0.00, A 0, B 0, C 0} C_DIS
LIN {X 98.26, Y 257.88, Z 0.00, A 0, B 0, C 0} C_DIS
LIN {X 98.47, Y 257.88, Z 0.00, A 0, B 0, C 0} C_DIS
LIN {X 98.69, Y 257.88, Z 0.00, A 0, B 0, C 0} C_DIS
LIN {X 98.91, Y 257.88, Z 0.00, A 0, B 0, C 0} C_DIS
LIN {X 99.13, Y 257.88, Z 0.00, A 0, B 0, C 0} C_DIS
LIN {X 99.34, Y 257.88, Z 0.00, A 0, B 0, C 0} C_DIS
LIN {X 99.56, Y 257.88, Z 0.00, A 0, B 0, C 0} C_DIS
LIN {X 99.78, Y 257.88, Z 0.00, A 0, B 0, C 0} C_DIS
LIN {X 100.00, Y 257.88, Z 0.00, A 0, B 0, C 0} C_DIS
LIN {X 100.21, Y 257.88, Z 0.00, A 0, B 0, C 0} C_DIS
LIN {X 100.43, Y 257.88, Z 0.00, A 0, B 0, C 0} C_DIS
LIN {X 100.65, Y 257.88, Z 0.00, A 0, B 0, C 0} C_DIS
LIN {X 100.87, Y 257.88, Z 0.00, A 0, B 0, C 0} C_DIS
LIN {X 101.08, Y 257.87, Z 0.00, A 0, B 0, C 0} C_DIS
LIN {X 101.30, Y 257.84, Z 0.00, A 0, B 0, C 0} C_DIS
LIN {X 101.51, Y 257.80, Z 0.00, A 0, B 0, C 0} C_DIS
LIN {X 101.73, Y 257.73, Z 0.00, A 0, B 0, C 0} C_DIS
LIN {X 101.94, Y 257.64, Z 0.00, A 0, B 0, C 0} C_DIS
LIN {X 102.15, Y 257.54, Z 0.00, A 0, B 0, C 0} C_DIS
LIN {X 102.35, Y 257.44, Z 0.00, A 0, B 0, C 0} C_DIS
LIN {X 102.53, Y 257.27, Z 0.00, A 0, B 0, C 0} C_DIS
LIN {X 102.69, Y 257.04, Z 0.00, A 0, B 0, C 0} C_DIS
LIN {X 102.84, Y 256.80, Z 0.00, A 0, B 0, C 0} C_DIS
LIN {X 103.00, Y 256.57, Z 0.00, A 0, B 0, C 0} C_DIS
LIN {X 103.14, Y 256.33, Z 0.00, A 0, B 0, C 0} C_DIS
LIN {X 103.21, Y 256.03, Z 0.00, A 0, B 0, C 0} C_DIS
LIN {X 103.24, Y 255.70, Z 0.00, A 0, B 0, C 0} C_DIS
LIN {X 103.25, Y 255.37, Z 0.00, A 0, B 0, C 0} C_DIS
LIN {X 103.22, Y 255.05, Z 0.00, A 0, B 0, C 0} C_DIS
LIN {X 103.15, Y 254.74, Z 0.00, A 0, B 0, C 0} C_DIS
LIN {X 103.05, Y 254.45, Z 0.00, A 0, B 0, C 0} C_DIS
LIN {X 102.93, Y 254.18, Z 0.00, A 0, B 0, C 0} C_DIS
LIN {X 102.79, Y 253.92, Z 0.00, A 0, B 0, C 0} C_DIS
LIN {X 102.64, Y 253.69, Z 0.00, A 0, B 0, C 0} C_DIS
LIN {X 102.47, Y 253.47, Z 0.00, A 0, B 0, C 0} C_DIS
LIN {X 102.30, Y 253.28, Z 0.00, A 0, B 0, C 0} C_DIS
LIN {X 102.11, Y 253.11, Z 0.00, A 0, B 0, C 0} C_DIS
LIN {X 101.92, Y 252.95, Z 0.00, A 0, B 0, C 0} C_DIS
LIN {X 101.74, Y 252.77, Z 0.00, A 0, B 0, C 0} C_DIS
LIN {X 101.57, Y 252.56, Z 0.00, A 0, B 0, C 0} C_DIS
LIN {X 101.41, Y 252.34, Z 0.00, A 0, B 0, C 0} C_DIS
LIN {X 101.25, Y 252.12, Z 0.00, A 0, B 0, C 0} C_DIS
LIN {X 101.09, Y 251.91, Z 0.00, A 0, B 0, C 0} C_DIS
LIN {X 100.92, Y 251.70, Z 0.00, A 0, B 0, C 0} C_DIS
LIN {X 100.75, Y 251.51, Z 0.00, A 0, B 0, C 0} C_DIS
LIN {X 100.56, Y 251.33, Z 0.00, A 0, B 0, C 0} C_DIS
LIN {X 100.38, Y 251.16, Z 0.00, A 0, B 0, C 0} C_DIS
LIN {X 100.18, Y 251.01, Z 0.00, A 0, B 0, C 0} C_DIS
LIN {X 99.98, Y 250.88, Z 0.00, A 0, B 0, C 0} C_DIS
LIN {X 99.78, Y 250.75, Z 0.00, A 0, B 0, C 0} C_DIS
LIN {X 99.60, Y 250.59, Z 0.00, A 0, B 0, C 0} C_DIS
LIN {X 99.41, Y 250.42, Z 0.00, A 0, B 0, C 0} C_DIS
LIN {X 99.21, Y 250.28, Z 0.00, A 0, B 0, C 0} C_DIS
LIN {X 99.01, Y 250.16, Z 0.00, A 0, B 0, C 0} C_DIS
LIN {X 98.82, Y 250.02, Z 0.00, A 0, B 0, C 0} C_DIS
LIN {X 98.63, Y 249.84, Z 0.00, A 0, B 0, C 0} C_DIS
LIN {X 98.44, Y 249.69, Z 0.00, A 0, B 0, C 0} C_DIS
LIN {X 98.24, Y 249.56, Z 0.00, A 0, B 0, C 0} C_DIS
LIN {X 98.04, Y 249.44, Z 0.00, A 0, B 0, C 0} C_DIS
LIN {X 97.85, Y 249.28, Z 0.00, A 0, B 0, C 0} C_DIS
LIN {X 97.67, Y 249.10, Z 0.00, A 0, B 0, C 0} C_DIS
LIN {X 97.47, Y 248.97, Z 0.00, A 0, B 0, C 0} C_DIS
LIN {X 97.27, Y 248.85, Z 0.00, A 0, B 0, C 0} C_DIS
LIN {X 97.07, Y 248.70, Z 0.00, A 0, B 0, C 0} C_DIS
LIN {X 96.89, Y 248.53, Z 0.00, A 0, B 0, C 0} C_DIS
LIN {X 96.70, Y 248.37, Z 0.00, A 0, B 0, C 0} C_DIS
LIN {X 96.50, Y 248.25, Z 0.00, A 0, B 0, C 0} C_DIS
LIN {X 96.30, Y 248.12, Z 0.00, A 0, B 0, C 0} C_DIS
LIN {X 96.11, Y 247.96, Z 0.00, A 0, B 0, C 0} C_DIS
LIN {X 95.92, Y 247.79, Z 0.00, A 0, B 0, C 0} C_DIS
LIN {X 95.73, Y 247.65, Z 0.00, A 0, B 0, C 0} C_DIS
LIN {X 95.52, Y 247.53, Z 0.00, A 0, B 0, C 0} C_DIS
LIN {X 95.33, Y 247.39, Z 0.00, A 0, B 0, C 0} C_DIS
LIN {X 95.14, Y 247.22, Z 0.00, A 0, B 0, C 0} C_DIS
LIN {X 94.95, Y 247.06, Z 0.00, A 0, B 0, C 0} C_DIS
LIN {X 94.75, Y 246.93, Z 0.00, A 0, B 0, C 0} C_DIS
LIN {X 94.55, Y 246.81, Z 0.00, A 0, B 0, C 0} C_DIS
LIN {X 94.36, Y 246.65, Z 0.00, A 0, B 0, C 0} C_DIS
LIN {X 94.18, Y 246.48, Z 0.00, A 0, B 0, C 0} C_DIS
LIN {X 93.99, Y 246.33, Z 0.00, A 0, B 0, C 0} C_DIS
LIN {X 93.78, Y 246.24, Z 0.00, A 0, B 0, C 0} C_DIS
LIN {X 93.56, Y 246.17, Z 0.00, A 0, B 0, C 0} C_DIS
LIN {X 93.36, Y 246.04, Z 0.00, A 0, B 0, C 0} C_DIS
LIN {X 93.16, Y 245.90, Z 0.00, A 0, B 0, C 0} C_DIS
LIN {X 92.96, Y 245.79, Z 0.00, A 0, B 0, C 0} C_DIS
LIN {X 92.75, Y 245.70, Z 0.00, A 0, B 0, C 0} C_DIS
LIN {X 92.55, Y 245.60, Z 0.00, A 0, B 0, C 0} C_DIS
LIN {X 92.34, Y 245.48, Z 0.00, A 0, B 0, C 0} C_DIS
LIN {X 92.16, Y 245.31, Z 0.00, A 0, B 0, C 0} C_DIS
LIN {X 91.97, Y 245.14, Z 0.00, A 0, B 0, C 0} C_DIS
LIN {X 91.77, Y 245.01, Z 0.00, A 0, B 0, C 0} C_DIS
LIN {X 91.57, Y 244.89, Z 0.00, A 0, B 0, C 0} C_DIS
LIN {X 91.38, Y 244.74, Z 0.00, A 0, B 0, C 0} C_DIS
LIN {X 91.19, Y 244.56, Z 0.00, A 0, B 0, C 0} C_DIS
LIN {X 91.00, Y 244.41, Z 0.00, A 0, B 0, C 0} C_DIS
LIN {X 90.80, Y 244.30, Z 0.00, A 0, B 0, C 0} C_DIS
LIN {X 90.61, Y 244.16, Z 0.00, A 0, B 0, C 0} C_DIS
LIN {X 90.43, Y 243.96, Z 0.00, A 0, B 0, C 0} C_DIS
LIN {X 90.28, Y 243.71, Z 0.00, A 0, B 0, C 0} C_DIS
LIN {X 90.17, Y 243.42, Z 0.00, A 0, B 0, C 0} C_DIS
LIN {X 90.12, Y 243.11, Z 0.00, A 0, B 0, C 0} C_DIS
LIN {X 90.13, Y 242.80, Z 0.00, A 0, B 0, C 0} C_DIS
LIN {X 90.16, Y 242.47, Z 0.00, A 0, B 0, C 0} C_DIS
LIN {X 90.22, Y 242.15, Z 0.00, A 0, B 0, C 0} C_DIS
LIN {X 90.31, Y 241.85, Z 0.00, A 0, B 0, C 0} C_DIS
LIN {X 90.41, Y 241.56, Z 0.00, A 0, B 0, C 0} C_DIS
LIN {X 90.52, Y 241.28, Z 0.00, A 0, B 0, C 0} C_DIS
LIN {X 90.61, Y 240.99, Z 0.00, A 0, B 0, C 0} C_DIS
LIN {X 90.70, Y 240.68, Z 0.00, A 0, B 0, C 0} C_DIS
LIN {X 90.79, Y 240.39, Z 0.00, A 0, B 0, C 0} C_DIS
LIN {X 90.90, Y 240.11, Z 0.00, A 0, B 0, C 0} C_DIS
LIN {X 91.01, Y 239.82, Z 0.00, A 0, B 0, C 0} C_DIS
LIN {X 91.10, Y 239.52, Z 0.00, A 0, B 0, C 0} C_DIS
LIN {X 91.18, Y 239.22, Z 0.00, A 0, B 0, C 0} C_DIS
LIN {X 91.28, Y 238.93, Z 0.00, A 0, B 0, C 0} C_DIS
LIN {X 91.39, Y 238.65, Z 0.00, A 0, B 0, C 0} C_DIS
LIN {X 91.49, Y 238.36, Z 0.00, A 0, B 0, C 0} C_DIS
LIN {X 91.57, Y 238.05, Z 0.00, A 0, B 0, C 0} C_DIS
LIN {X 91.66, Y 237.76, Z 0.00, A 0, B 0, C 0} C_DIS
LIN {X 91.77, Y 237.48, Z 0.00, A 0, B 0, C 0} C_DIS
LIN {X 91.88, Y 237.20, Z 0.00, A 0, B 0, C 0} C_DIS
LIN {X 91.97, Y 236.89, Z 0.00, A 0, B 0, C 0} C_DIS
LIN {X 92.05, Y 236.59, Z 0.00, A 0, B 0, C 0} C_DIS
LIN {X 92.15, Y 236.30, Z 0.00, A 0, B 0, C 0} C_DIS
LIN {X 92.27, Y 236.03, Z 0.00, A 0, B 0, C 0} C_DIS
LIN {X 92.36, Y 235.73, Z 0.00, A 0, B 0, C 0} C_DIS
LIN {X 92.44, Y 235.43, Z 0.00, A 0, B 0, C 0} C_DIS
LIN {X 92.53, Y 235.13, Z 0.00, A 0, B 0, C 0} C_DIS
LIN {X 92.65, Y 234.85, Z 0.00, A 0, B 0, C 0} C_DIS
LIN {X 92.75, Y 234.57, Z 0.00, A 0, B 0, C 0} C_DIS
LIN {X 92.84, Y 234.27, Z 0.00, A 0, B 0, C 0} C_DIS
LIN {X 92.92, Y 233.96, Z 0.00, A 0, B 0, C 0} C_DIS
LIN {X 93.02, Y 233.67, Z 0.00, A 0, B 0, C 0} C_DIS
LIN {X 93.14, Y 233.40, Z 0.00, A 0, B 0, C 0} C_DIS
LIN {X 93.23, Y 233.10, Z 0.00, A 0, B 0, C 0} C_DIS
LIN {X 93.31, Y 232.80, Z 0.00, A 0, B 0, C 0} C_DIS
LIN {X 93.40, Y 232.50, Z 0.00, A 0, B 0, C 0} C_DIS
LIN {X 93.52, Y 232.22, Z 0.00, A 0, B 0, C 0} C_DIS
LIN {X 93.63, Y 231.94, Z 0.00, A 0, B 0, C 0} C_DIS
LIN {X 93.71, Y 231.64, Z 0.00, A 0, B 0, C 0} C_DIS
LIN {X 93.79, Y 231.33, Z 0.00, A 0, B 0, C 0} C_DIS
LIN {X 93.89, Y 231.05, Z 0.00, A 0, B 0, C 0} C_DIS
LIN {X 94.01, Y 230.77, Z 0.00, A 0, B 0, C 0} C_DIS
LIN {X 94.10, Y 230.48, Z 0.00, A 0, B 0, C 0} C_DIS
LIN {X 94.18, Y 230.17, Z 0.00, A 0, B 0, C 0} C_DIS
LIN {X 94.28, Y 229.87, Z 0.00, A 0, B 0, C 0} C_DIS
LIN {X 94.39, Y 229.60, Z 0.00, A 0, B 0, C 0} C_DIS
LIN {X 94.49, Y 229.31, Z 0.00, A 0, B 0, C 0} C_DIS
LIN {X 94.58, Y 229.00, Z 0.00, A 0, B 0, C 0} C_DIS
LIN {X 94.67, Y 228.71, Z 0.00, A 0, B 0, C 0} C_DIS
LIN {X 94.77, Y 228.42, Z 0.00, A 0, B 0, C 0} C_DIS
LIN {X 94.88, Y 228.14, Z 0.00, A 0, B 0, C 0} C_DIS
LIN {X 94.98, Y 227.85, Z 0.00, A 0, B 0, C 0} C_DIS
LIN {X 95.05, Y 227.54, Z 0.00, A 0, B 0, C 0} C_DIS
LIN {X 95.10, Y 227.22, Z 0.00, A 0, B 0, C 0} C_DIS
LIN {X 95.17, Y 226.91, Z 0.00, A 0, B 0, C 0} C_DIS
LIN {X 95.26, Y 226.61, Z 0.00, A 0, B 0, C 0} C_DIS
LIN {X 95.35, Y 226.31, Z 0.00, A 0, B 0, C 0} C_DIS
LIN {X 95.41, Y 226.00, Z 0.00, A 0, B 0, C 0} C_DIS
LIN {X 95.46, Y 225.68, Z 0.00, A 0, B 0, C 0} C_DIS
LIN {X 95.51, Y 225.36, Z 0.00, A 0, B 0, C 0} C_DIS
LIN {X 95.58, Y 225.05, Z 0.00, A 0, B 0, C 0} C_DIS
LIN {X 95.66, Y 224.75, Z 0.00, A 0, B 0, C 0} C_DIS
LIN {X 95.76, Y 224.45, Z 0.00, A 0, B 0, C 0} C_DIS
LIN {X 95.83, Y 224.14, Z 0.00, A 0, B 0, C 0} C_DIS
LIN {X 95.88, Y 223.83, Z 0.00, A 0, B 0, C 0} C_DIS
LIN {X 95.92, Y 223.50, Z 0.00, A 0, B 0, C 0} C_DIS
LIN {X 95.99, Y 223.19, Z 0.00, A 0, B 0, C 0} C_DIS
LIN {X 96.08, Y 222.89, Z 0.00, A 0, B 0, C 0} C_DIS
LIN {X 96.16, Y 222.59, Z 0.00, A 0, B 0, C 0} C_DIS
LIN {X 96.23, Y 222.28, Z 0.00, A 0, B 0, C 0} C_DIS
LIN {X 96.29, Y 221.97, Z 0.00, A 0, B 0, C 0} C_DIS
LIN {X 96.35, Y 221.65, Z 0.00, A 0, B 0, C 0} C_DIS
LIN {X 96.41, Y 221.33, Z 0.00, A 0, B 0, C 0} C_DIS
LIN {X 96.46, Y 221.02, Z 0.00, A 0, B 0, C 0} C_DIS
LIN {X 96.51, Y 220.69, Z 0.00, A 0, B 0, C 0} C_DIS
LIN {X 96.53, Y 220.37, Z 0.00, A 0, B 0, C 0} C_DIS
LIN {X 96.55, Y 220.04, Z 0.00, A 0, B 0, C 0} C_DIS
LIN {X 96.55, Y 219.72, Z 0.00, A 0, B 0, C 0} C_DIS
LIN {X 96.56, Y 219.39, Z 0.00, A 0, B 0, C 0} C_DIS
LIN {X 96.58, Y 219.06, Z 0.00, A 0, B 0, C 0} C_DIS
LIN {X 96.61, Y 218.74, Z 0.00, A 0, B 0, C 0} C_DIS
LIN {X 96.66, Y 218.42, Z 0.00, A 0, B 0, C 0} C_DIS
LIN {X 96.71, Y 218.10, Z 0.00, A 0, B 0, C 0} C_DIS
LIN {X 96.77, Y 217.79, Z 0.00, A 0, B 0, C 0} C_DIS
LIN {X 96.83, Y 217.47, Z 0.00, A 0, B 0, C 0} C_DIS
LIN {X 96.89, Y 217.15, Z 0.00, A 0, B 0, C 0} C_DIS
LIN {X 96.93, Y 216.83, Z 0.00, A 0, B 0, C 0} C_DIS
LIN {X 96.96, Y 216.51, Z 0.00, A 0, B 0, C 0} C_DIS
LIN {X 96.98, Y 216.18, Z 0.00, A 0, B 0, C 0} C_DIS
LIN {X 96.99, Y 215.86, Z 0.00, A 0, B 0, C 0} C_DIS
LIN {X 97.00, Y 215.53, Z 0.00, A 0, B 0, C 0} C_DIS
LIN {X 97.01, Y 215.20, Z 0.00, A 0, B 0, C 0} C_DIS
LIN {X 97.04, Y 214.88, Z 0.00, A 0, B 0, C 0} C_DIS
LIN {X 97.08, Y 214.56, Z 0.00, A 0, B 0, C 0} C_DIS
LIN {X 97.13, Y 214.24, Z 0.00, A 0, B 0, C 0} C_DIS
LIN {X 97.20, Y 213.92, Z 0.00, A 0, B 0, C 0} C_DIS
LIN {X 97.26, Y 213.61, Z 0.00, A 0, B 0, C 0} C_DIS
LIN {X 97.32, Y 213.29, Z 0.00, A 0, B 0, C 0} C_DIS
LIN {X 97.36, Y 212.97, Z 0.00, A 0, B 0, C 0} C_DIS
LIN {X 97.39, Y 212.65, Z 0.00, A 0, B 0, C 0} C_DIS
LIN {X 97.41, Y 212.32, Z 0.00, A 0, B 0, C 0} C_DIS
LIN {X 97.42, Y 212.00, Z 0.00, A 0, B 0, C 0} C_DIS
LIN {X 97.43, Y 211.67, Z 0.00, A 0, B 0, C 0} C_DIS
LIN {X 97.43, Y 211.34, Z 0.00, A 0, B 0, C 0} C_DIS
LIN {X 97.43, Y 211.01, Z 0.00, A 0, B 0, C 0} C_DIS
LIN {X 97.42, Y 210.68, Z 0.00, A 0, B 0, C 0} C_DIS
LIN {X 97.42, Y 210.36, Z 0.00, A 0, B 0, C 0} C_DIS
LIN {X 97.42, Y 210.03, Z 0.00, A 0, B 0, C 0} C_DIS
LIN {X 97.42, Y 209.70, Z 0.00, A 0, B 0, C 0} C_DIS
LIN {X 97.42, Y 209.37, Z 0.00, A 0, B 0, C 0} C_DIS
LIN {X 97.42, Y 209.05, Z 0.00, A 0, B 0, C 0} C_DIS
LIN {X 97.42, Y 208.72, Z 0.00, A 0, B 0, C 0} C_DIS
LIN {X 97.43, Y 208.39, Z 0.00, A 0, B 0, C 0} C_DIS
LIN {X 97.43, Y 208.06, Z 0.00, A 0, B 0, C 0} C_DIS
LIN {X 97.43, Y 207.73, Z 0.00, A 0, B 0, C 0} C_DIS
LIN {X 97.43, Y 207.41, Z 0.00, A 0, B 0, C 0} C_DIS
LIN {X 97.43, Y 207.08, Z 0.00, A 0, B 0, C 0} C_DIS
LIN {X 97.42, Y 206.75, Z 0.00, A 0, B 0, C 0} C_DIS
LIN {X 97.41, Y 206.42, Z 0.00, A 0, B 0, C 0} C_DIS
LIN {X 97.39, Y 206.10, Z 0.00, A 0, B 0, C 0} C_DIS
LIN {X 97.37, Y 205.78, Z 0.00, A 0, B 0, C 0} C_DIS
LIN {X 97.33, Y 205.45, Z 0.00, A 0, B 0, C 0} C_DIS
LIN {X 97.28, Y 205.14, Z 0.00, A 0, B 0, C 0} C_DIS
LIN {X 97.22, Y 204.82, Z 0.00, A 0, B 0, C 0} C_DIS
LIN {X 97.16, Y 204.50, Z 0.00, A 0, B 0, C 0} C_DIS
LIN {X 97.10, Y 204.19, Z 0.00, A 0, B 0, C 0} C_DIS
LIN {X 97.05, Y 203.87, Z 0.00, A 0, B 0, C 0} C_DIS
LIN {X 97.01, Y 203.54, Z 0.00, A 0, B 0, C 0} C_DIS
LIN {X 96.99, Y 203.22, Z 0.00, A 0, B 0, C 0} C_DIS
LIN {X 96.98, Y 202.89, Z 0.00, A 0, B 0, C 0} C_DIS
LIN {X 96.99, Y 202.56, Z 0.00, A 0, B 0, C 0} C_DIS
LIN {X 97.00, Y 202.23, Z 0.00, A 0, B 0, C 0} C_DIS
LIN {X 97.00, Y 201.91, Z 0.00, A 0, B 0, C 0} C_DIS
LIN {X 96.98, Y 201.58, Z 0.00, A 0, B 0, C 0} C_DIS
LIN {X 96.94, Y 201.26, Z 0.00, A 0, B 0, C 0} C_DIS
LIN {X 96.90, Y 200.94, Z 0.00, A 0, B 0, C 0} C_DIS
LIN {X 96.84, Y 200.62, Z 0.00, A 0, B 0, C 0} C_DIS
LIN {X 96.79, Y 200.30, Z 0.00, A 0, B 0, C 0} C_DIS
LIN {X 96.74, Y 199.98, Z 0.00, A 0, B 0, C 0} C_DIS
LIN {X 96.69, Y 199.66, Z 0.00, A 0, B 0, C 0} C_DIS
LIN {X 96.64, Y 199.35, Z 0.00, A 0, B 0, C 0} C_DIS
LIN {X 96.58, Y 199.03, Z 0.00, A 0, B 0, C 0} C_DIS
LIN {X 96.53, Y 198.71, Z 0.00, A 0, B 0, C 0} C_DIS
LIN {X 96.48, Y 198.39, Z 0.00, A 0, B 0, C 0} C_DIS
LIN {X 96.42, Y 198.08, Z 0.00, A 0, B 0, C 0} C_DIS
LIN {X 96.37, Y 197.76, Z 0.00, A 0, B 0, C 0} C_DIS
LIN {X 96.32, Y 197.44, Z 0.00, A 0, B 0, C 0} C_DIS
LIN {X 96.26, Y 197.12, Z 0.00, A 0, B 0, C 0} C_DIS
LIN {X 96.21, Y 196.81, Z 0.00, A 0, B 0, C 0} C_DIS
LIN {X 96.16, Y 196.49, Z 0.00, A 0, B 0, C 0} C_DIS
LIN {X 96.10, Y 196.17, Z 0.00, A 0, B 0, C 0} C_DIS
LIN {X 96.05, Y 195.85, Z 0.00, A 0, B 0, C 0} C_DIS
LIN {X 96.01, Y 195.53, Z 0.00, A 0, B 0, C 0} C_DIS
LIN {X 95.96, Y 195.21, Z 0.00, A 0, B 0, C 0} C_DIS
LIN {X 95.90, Y 194.89, Z 0.00, A 0, B 0, C 0} C_DIS
LIN {X 95.84, Y 194.58, Z 0.00, A 0, B 0, C 0} C_DIS
LIN {X 95.77, Y 194.27, Z 0.00, A 0, B 0, C 0} C_DIS
LIN {X 95.69, Y 193.97, Z 0.00, A 0, B 0, C 0} C_DIS
LIN {X 95.61, Y 193.67, Z 0.00, A 0, B 0, C 0} C_DIS
LIN {X 95.54, Y 193.36, Z 0.00, A 0, B 0, C 0} C_DIS
LIN {X 95.48, Y 193.04, Z 0.00, A 0, B 0, C 0} C_DIS
LIN {X 95.41, Y 192.73, Z 0.00, A 0, B 0, C 0} C_DIS
LIN {X 95.31, Y 192.44, Z 0.00, A 0, B 0, C 0} C_DIS
LIN {X 95.19, Y 192.17, Z 0.00, A 0, B 0, C 0} C_DIS
LIN {X 95.09, Y 191.87, Z 0.00, A 0, B 0, C 0} C_DIS
LIN {X 95.03, Y 191.56, Z 0.00, A 0, B 0, C 0} C_DIS
LIN {X 94.96, Y 191.25, Z 0.00, A 0, B 0, C 0} C_DIS
LIN {X 94.88, Y 190.94, Z 0.00, A 0, B 0, C 0} C_DIS
LIN {X 94.80, Y 190.64, Z 0.00, A 0, B 0, C 0} C_DIS
LIN {X 94.73, Y 190.34, Z 0.00, A 0, B 0, C 0} C_DIS
LIN {X 94.66, Y 190.02, Z 0.00, A 0, B 0, C 0} C_DIS
LIN {X 94.60, Y 189.71, Z 0.00, A 0, B 0, C 0} C_DIS
LIN {X 94.52, Y 189.40, Z 0.00, A 0, B 0, C 0} C_DIS
LIN {X 94.43, Y 189.11, Z 0.00, A 0, B 0, C 0} C_DIS
LIN {X 94.31, Y 188.84, Z 0.00, A 0, B 0, C 0} C_DIS
LIN {X 94.21, Y 188.55, Z 0.00, A 0, B 0, C 0} C_DIS
LIN {X 94.13, Y 188.24, Z 0.00, A 0, B 0, C 0} C_DIS
LIN {X 94.04, Y 187.94, Z 0.00, A 0, B 0, C 0} C_DIS
LIN {X 93.93, Y 187.66, Z 0.00, A 0, B 0, C 0} C_DIS
LIN {X 93.82, Y 187.38, Z 0.00, A 0, B 0, C 0} C_DIS
LIN {X 93.73, Y 187.08, Z 0.00, A 0, B 0, C 0} C_DIS
LIN {X 93.64, Y 186.78, Z 0.00, A 0, B 0, C 0} C_DIS
LIN {X 93.55, Y 186.49, Z 0.00, A 0, B 0, C 0} C_DIS
LIN {X 93.44, Y 186.20, Z 0.00, A 0, B 0, C 0} C_DIS
LIN {X 93.32, Y 185.93, Z 0.00, A 0, B 0, C 0} C_DIS
LIN {X 93.20, Y 185.66, Z 0.00, A 0, B 0, C 0} C_DIS
LIN {X 93.07, Y 185.39, Z 0.00, A 0, B 0, C 0} C_DIS
LIN {X 92.94, Y 185.13, Z 0.00, A 0, B 0, C 0} C_DIS
LIN {X 92.82, Y 184.86, Z 0.00, A 0, B 0, C 0} C_DIS
LIN {X 92.70, Y 184.58, Z 0.00, A 0, B 0, C 0} C_DIS
LIN {X 92.59, Y 184.30, Z 0.00, A 0, B 0, C 0} C_DIS
LIN {X 92.50, Y 184.01, Z 0.00, A 0, B 0, C 0} C_DIS
LIN {X 92.41, Y 183.71, Z 0.00, A 0, B 0, C 0} C_DIS
LIN {X 92.31, Y 183.41, Z 0.00, A 0, B 0, C 0} C_DIS
LIN {X 92.21, Y 183.13, Z 0.00, A 0, B 0, C 0} C_DIS
LIN {X 92.09, Y 182.85, Z 0.00, A 0, B 0, C 0} C_DIS
LIN {X 91.98, Y 182.57, Z 0.00, A 0, B 0, C 0} C_DIS
LIN {X 91.85, Y 182.30, Z 0.00, A 0, B 0, C 0} C_DIS
LIN {X 91.72, Y 182.05, Z 0.00, A 0, B 0, C 0} C_DIS
LIN {X 91.57, Y 181.81, Z 0.00, A 0, B 0, C 0} C_DIS
LIN {X 91.42, Y 181.58, Z 0.00, A 0, B 0, C 0} C_DIS
LIN {X 91.27, Y 181.33, Z 0.00, A 0, B 0, C 0} C_DIS
LIN {X 91.15, Y 181.07, Z 0.00, A 0, B 0, C 0} C_DIS
LIN {X 91.03, Y 180.79, Z 0.00, A 0, B 0, C 0} C_DIS
LIN {X 90.91, Y 180.51, Z 0.00, A 0, B 0, C 0} C_DIS
LIN {X 90.80, Y 180.23, Z 0.00, A 0, B 0, C 0} C_DIS
LIN {X 90.68, Y 179.96, Z 0.00, A 0, B 0, C 0} C_DIS
LIN {X 90.55, Y 179.69, Z 0.00, A 0, B 0, C 0} C_DIS
LIN {X 90.41, Y 179.44, Z 0.00, A 0, B 0, C 0} C_DIS
LIN {X 90.27, Y 179.20, Z 0.00, A 0, B 0, C 0} C_DIS
LIN {X 90.12, Y 178.97, Z 0.00, A 0, B 0, C 0} C_DIS
LIN {X 89.96, Y 178.73, Z 0.00, A 0, B 0, C 0} C_DIS
LIN {X 89.81, Y 178.50, Z 0.00, A 0, B 0, C 0} C_DIS
LIN {X 89.66, Y 178.26, Z 0.00, A 0, B 0, C 0} C_DIS
LIN {X 89.52, Y 178.01, Z 0.00, A 0, B 0, C 0} C_DIS
LIN {X 89.39, Y 177.76, Z 0.00, A 0, B 0, C 0} C_DIS
LIN {X 89.27, Y 177.49, Z 0.00, A 0, B 0, C 0} C_DIS
LIN {X 89.15, Y 177.21, Z 0.00, A 0, B 0, C 0} C_DIS
LIN {X 89.04, Y 176.93, Z 0.00, A 0, B 0, C 0} C_DIS
LIN {X 88.92, Y 176.65, Z 0.00, A 0, B 0, C 0} C_DIS
LIN {X 88.80, Y 176.38, Z 0.00, A 0, B 0, C 0} C_DIS
LIN {X 88.67, Y 176.11, Z 0.00, A 0, B 0, C 0} C_DIS
LIN {X 88.55, Y 175.84, Z 0.00, A 0, B 0, C 0} C_DIS
LIN {X 88.46, Y 175.55, Z 0.00, A 0, B 0, C 0} C_DIS
LIN {X 88.38, Y 175.24, Z 0.00, A 0, B 0, C 0} C_DIS
LIN {X 88.34, Y 174.92, Z 0.00, A 0, B 0, C 0} C_DIS
LIN {X 88.32, Y 174.59, Z 0.00, A 0, B 0, C 0} C_DIS
LIN {X 88.33, Y 174.25, Z 0.00, A 0, B 0, C 0} C_DIS
LIN {X 88.37, Y 173.93, Z 0.00, A 0, B 0, C 0} C_DIS
LIN {X 88.45, Y 173.62, Z 0.00, A 0, B 0, C 0} C_DIS
LIN {X 88.55, Y 173.34, Z 0.00, A 0, B 0, C 0} C_DIS
LIN {X 88.67, Y 173.07, Z 0.00, A 0, B 0, C 0} C_DIS
LIN {X 88.81, Y 172.82, Z 0.00, A 0, B 0, C 0} C_DIS
LIN {X 88.95, Y 172.58, Z 0.00, A 0, B 0, C 0} C_DIS
LIN {X 89.11, Y 172.35, Z 0.00, A 0, B 0, C 0} C_DIS
LIN {X 89.27, Y 172.12, Z 0.00, A 0, B 0, C 0} C_DIS
LIN {X 89.42, Y 171.88, Z 0.00, A 0, B 0, C 0} C_DIS
LIN {X 89.57, Y 171.65, Z 0.00, A 0, B 0, C 0} C_DIS
LIN {X 89.73, Y 171.42, Z 0.00, A 0, B 0, C 0} C_DIS
LIN {X 89.88, Y 171.19, Z 0.00, A 0, B 0, C 0} C_DIS
LIN {X 90.03, Y 170.96, Z 0.00, A 0, B 0, C 0} C_DIS
LIN {X 90.19, Y 170.73, Z 0.00, A 0, B 0, C 0} C_DIS
LIN {X 90.34, Y 170.50, Z 0.00, A 0, B 0, C 0} C_DIS
LIN {X 90.50, Y 170.27, Z 0.00, A 0, B 0, C 0} C_DIS
LIN {X 90.65, Y 170.04, Z 0.00, A 0, B 0, C 0} C_DIS
LIN {X 90.80, Y 169.80, Z 0.00, A 0, B 0, C 0} C_DIS
LIN {X 90.96, Y 169.57, Z 0.00, A 0, B 0, C 0} C_DIS
LIN {X 91.11, Y 169.34, Z 0.00, A 0, B 0, C 0} C_DIS
LIN {X 91.27, Y 169.11, Z 0.00, A 0, B 0, C 0} C_DIS
LIN {X 91.42, Y 168.88, Z 0.00, A 0, B 0, C 0} C_DIS
LIN {X 91.57, Y 168.64, Z 0.00, A 0, B 0, C 0} C_DIS
LIN {X 91.73, Y 168.41, Z 0.00, A 0, B 0, C 0} C_DIS
LIN {X 91.88, Y 168.18, Z 0.00, A 0, B 0, C 0} C_DIS
LIN {X 92.03, Y 167.95, Z 0.00, A 0, B 0, C 0} C_DIS
LIN {X 92.19, Y 167.71, Z 0.00, A 0, B 0, C 0} C_DIS
LIN {X 92.34, Y 167.48, Z 0.00, A 0, B 0, C 0} C_DIS
LIN {X 92.49, Y 167.25, Z 0.00, A 0, B 0, C 0} C_DIS
LIN {X 92.65, Y 167.02, Z 0.00, A 0, B 0, C 0} C_DIS
LIN {X 92.80, Y 166.79, Z 0.00, A 0, B 0, C 0} C_DIS
LIN {X 92.96, Y 166.56, Z 0.00, A 0, B 0, C 0} C_DIS
LIN {X 93.11, Y 166.33, Z 0.00, A 0, B 0, C 0} C_DIS
LIN {X 93.27, Y 166.11, Z 0.00, A 0, B 0, C 0} C_DIS
LIN {X 93.44, Y 165.91, Z 0.00, A 0, B 0, C 0} C_DIS
LIN {X 93.63, Y 165.74, Z 0.00, A 0, B 0, C 0} C_DIS
LIN {X 93.83, Y 165.62, Z 0.00, A 0, B 0, C 0} C_DIS
LIN {X 94.05, Y 165.54, Z 0.00, A 0, B 0, C 0} C_DIS
LIN {X 94.26, Y 165.51, Z 0.00, A 0, B 0, C 0} C_DIS
LIN {X 94.48, Y 165.54, Z 0.00, A 0, B 0, C 0} C_DIS
LIN {X 94.69, Y 165.62, Z 0.00, A 0, B 0, C 0} C_DIS
LIN {X 94.89, Y 165.76, Z 0.00, A 0, B 0, C 0} C_DIS
LIN {X 95.06, Y 165.95, Z 0.00, A 0, B 0, C 0} C_DIS
LIN {X 95.21, Y 166.19, Z 0.00, A 0, B 0, C 0} C_DIS
LIN {X 95.34, Y 166.46, Z 0.00, A 0, B 0, C 0} C_DIS
LIN {X 95.46, Y 166.73, Z 0.00, A 0, B 0, C 0} C_DIS
LIN {X 95.60, Y 166.99, Z 0.00, A 0, B 0, C 0} C_DIS
LIN {X 95.73, Y 167.23, Z 0.00, A 0, B 0, C 0} C_DIS
LIN {X 95.88, Y 167.47, Z 0.00, A 0, B 0, C 0} C_DIS
LIN {X 96.03, Y 167.71, Z 0.00, A 0, B 0, C 0} C_DIS
LIN {X 96.19, Y 167.94, Z 0.00, A 0, B 0, C 0} C_DIS
LIN {X 96.34, Y 168.17, Z 0.00, A 0, B 0, C 0} C_DIS
LIN {X 96.50, Y 168.39, Z 0.00, A 0, B 0, C 0} C_DIS
LIN {X 96.66, Y 168.62, Z 0.00, A 0, B 0, C 0} C_DIS
LIN {X 96.81, Y 168.85, Z 0.00, A 0, B 0, C 0} C_DIS
LIN {X 96.96, Y 169.09, Z 0.00, A 0, B 0, C 0} C_DIS
LIN {X 97.11, Y 169.32, Z 0.00, A 0, B 0, C 0} C_DIS
LIN {X 97.26, Y 169.56, Z 0.00, A 0, B 0, C 0} C_DIS
LIN {X 97.40, Y 169.81, Z 0.00, A 0, B 0, C 0} C_DIS
LIN {X 97.53, Y 170.07, Z 0.00, A 0, B 0, C 0} C_DIS
LIN {X 97.66, Y 170.34, Z 0.00, A 0, B 0, C 0} C_DIS
LIN {X 97.77, Y 170.62, Z 0.00, A 0, B 0, C 0} C_DIS
LIN {X 97.89, Y 170.90, Z 0.00, A 0, B 0, C 0} C_DIS
LIN {X 98.00, Y 171.18, Z 0.00, A 0, B 0, C 0} C_DIS
LIN {X 98.12, Y 171.45, Z 0.00, A 0, B 0, C 0} C_DIS
LIN {X 98.26, Y 171.70, Z 0.00, A 0, B 0, C 0} C_DIS
